Fanuc TP program (LS listing): btu_logo.ls

/PROG  btu_logo
/ATTR
COMMENT	= "19-03-22 13:07:40";
PROG_SIZE	= 0;
DEFAULT_GROUP	= 1, *, *, *, *;
/APPL
    ARC Welding Equipment: 1, *, *, *, *;
/MN
   1:  CALL HOME_ALL;
   1:  UFRAME_NUM = 1;
   1:  UTOOL_NUM = 3;
   1:  COL GUARD ADJUST 150;
   1:  MESSAGE[- Layer/Ebene 1];
   1:  PR[91] = PR[90];
   1:  GO[2]=3;
   1:  PR[91,1] = PR[90,1] + 3.907;
   1:  PR[91,2] = PR[90,2] + 46.803;
   1:  PR[91,3] = PR[90,3] + 2.795;
   1:  MESSAGE[Teach Startpoint in PR91];
   1:  MESSAGE[Weld speed R100 in mm/sec];
   1:  MESSAGE[Retraction +Z in R101 in mm];
   1:  MESSAGE[Retraction speed in R102 in %];
   1:  PR[92] = PR[91];
   1:  PR[92,3] = PR[92,3] + R[101];
   1:J PR[92] R[102]% CNT100;
   1:L PR[91] 100mm/sec CNT100 RampTo R[100];
   1:  PR[91,1] = PR[90,1] + 3.583;
   1:  PR[91,2] = PR[90,2] + 46.861;
   1:L PR[91] R[100]mm/sec CNT100;
   1:  PR[91,1] = PR[90,1] + 3.247;
   1:  PR[91,2] = PR[90,2] + 46.900;
   1:L PR[91] R[100]mm/sec CNT100;
   1:  PR[91,1] = PR[90,1] + 2.612;
   1:  PR[91,2] = PR[90,2] + 47.029;
   1:L PR[91] R[100]mm/sec CNT100;
   1:  PR[91,1] = PR[90,1] + 1.805;
   1:  PR[91,2] = PR[90,2] + 47.067;
   1:L PR[91] R[100]mm/sec CNT100;
   1:  PR[91,1] = PR[90,1] + 1.782;
   1:  PR[91,2] = PR[90,2] + 47.066;
   1:L PR[91] R[100]mm/sec CNT100;
   1:  PR[91,1] = PR[90,1] + 1.030;
   1:  PR[91,2] = PR[90,2] + 46.980;
   1:L PR[91] R[100]mm/sec CNT100;
   1:  PR[91,1] = PR[90,1] + 0.258;
   1:  PR[91,2] = PR[90,2] + 46.814;
   1:L PR[91] R[100]mm/sec CNT100;
   1:  PR[91,1] = PR[90,1] + -0.573;
   1:  PR[91,2] = PR[90,2] + 46.433;
   1:L PR[91] R[100]mm/sec CNT100;
   1:  PR[91,1] = PR[90,1] + -0.582;
   1:  PR[91,2] = PR[90,2] + 46.430;
   1:L PR[91] R[100]mm/sec CNT100;
   1:  PR[91,1] = PR[90,1] + -1.294;
   1:  PR[91,2] = PR[90,2] + 45.950;
   1:L PR[91] R[100]mm/sec CNT100;
   1:  PR[91,1] = PR[90,1] + -1.634;
   1:  PR[91,2] = PR[90,2] + 45.636;
   1:L PR[91] R[100]mm/sec CNT100;
   1:  PR[91,1] = PR[90,1] + -2.312;
   1:  PR[91,2] = PR[90,2] + 44.852;
   1:L PR[91] R[100]mm/sec CNT100;
   1:  PR[91,1] = PR[90,1] + -2.541;
   1:  PR[91,2] = PR[90,2] + 44.349;
   1:L PR[91] R[100]mm/sec CNT100;
   1:  PR[91,1] = PR[90,1] + -2.727;
   1:  PR[91,2] = PR[90,2] + 43.996;
   1:L PR[91] R[100]mm/sec CNT100;
   1:  PR[91,1] = PR[90,1] + -3.065;
   1:  PR[91,2] = PR[90,2] + 43.254;
   1:L PR[91] R[100]mm/sec CNT100;
   1:  PR[91,1] = PR[90,1] + -3.083;
   1:  PR[91,2] = PR[90,2] + 43.063;
   1:L PR[91] R[100]mm/sec CNT100;
   1:  PR[91,1] = PR[90,1] + -3.240;
   1:  PR[91,2] = PR[90,2] + 42.434;
   1:L PR[91] R[100]mm/sec CNT100;
   1:  PR[91,1] = PR[90,1] + -3.248;
   1:  PR[91,2] = PR[90,2] + 42.049;
   1:L PR[91] R[100]mm/sec CNT100;
   1:  PR[91,1] = PR[90,1] + -3.284;
   1:  PR[91,2] = PR[90,2] + 41.564;
   1:L PR[91] R[100]mm/sec CNT100;
   1:  PR[91,1] = PR[90,1] + -3.289;
   1:  PR[91,2] = PR[90,2] + 40.607;
   1:L PR[91] R[100]mm/sec CNT100;
   1:  PR[91,1] = PR[90,1] + -3.286;
   1:  PR[91,2] = PR[90,2] + 2.178;
   1:L PR[91] R[100]mm/sec CNT100;
   1:  PR[91,1] = PR[90,1] + -3.273;
   1:  PR[91,2] = PR[90,2] + 1.199;
   1:L PR[91] R[100]mm/sec CNT100;
   1:  PR[91,1] = PR[90,1] + -3.212;
   1:  PR[91,2] = PR[90,2] + -0.213;
   1:L PR[91] R[100]mm/sec CNT100;
   1:  PR[91,1] = PR[90,1] + -3.152;
   1:  PR[91,2] = PR[90,2] + -0.737;
   1:L PR[91] R[100]mm/sec CNT100;
   1:  PR[91,1] = PR[90,1] + -3.131;
   1:  PR[91,2] = PR[90,2] + -1.080;
   1:L PR[91] R[100]mm/sec CNT100;
   1:  PR[91,1] = PR[90,1] + -3.026;
   1:  PR[91,2] = PR[90,2] + -1.687;
   1:L PR[91] R[100]mm/sec CNT100;
   1:  PR[91,1] = PR[90,1] + -3.009;
   1:  PR[91,2] = PR[90,2] + -1.889;
   1:L PR[91] R[100]mm/sec CNT100;
   1:  PR[91,1] = PR[90,1] + -2.860;
   1:  PR[91,2] = PR[90,2] + -2.483;
   1:L PR[91] R[100]mm/sec CNT100;
   1:  PR[91,1] = PR[90,1] + -2.816;
   1:  PR[91,2] = PR[90,2] + -2.594;
   1:L PR[91] R[100]mm/sec CNT100;
   1:  PR[91,1] = PR[90,1] + -2.568;
   1:  PR[91,2] = PR[90,2] + -3.464;
   1:L PR[91] R[100]mm/sec CNT100;
   1:  PR[91,1] = PR[90,1] + -2.555;
   1:  PR[91,2] = PR[90,2] + -3.686;
   1:L PR[91] R[100]mm/sec CNT100;
   1:  PR[91,1] = PR[90,1] + -2.415;
   1:  PR[91,2] = PR[90,2] + -4.292;
   1:L PR[91] R[100]mm/sec CNT100;
   1:  PR[91,1] = PR[90,1] + -2.298;
   1:  PR[91,2] = PR[90,2] + -5.127;
   1:L PR[91] R[100]mm/sec CNT100;
   1:  PR[91,1] = PR[90,1] + -2.153;
   1:  PR[91,2] = PR[90,2] + -5.601;
   1:L PR[91] R[100]mm/sec CNT100;
   1:  PR[91,1] = PR[90,1] + -2.125;
   1:  PR[91,2] = PR[90,2] + -5.801;
   1:L PR[91] R[100]mm/sec CNT100;
   1:  PR[91,1] = PR[90,1] + -1.883;
   1:  PR[91,2] = PR[90,2] + -6.260;
   1:L PR[91] R[100]mm/sec CNT100;
   1:  PR[91,1] = PR[90,1] + -1.467;
   1:  PR[91,2] = PR[90,2] + -7.196;
   1:L PR[91] R[100]mm/sec CNT100;
   1:  PR[91,1] = PR[90,1] + -1.390;
   1:  PR[91,2] = PR[90,2] + -7.658;
   1:L PR[91] R[100]mm/sec CNT100;
   1:  PR[91,1] = PR[90,1] + -1.315;
   1:  PR[91,2] = PR[90,2] + -7.984;
   1:L PR[91] R[100]mm/sec CNT100;
   1:  PR[91,1] = PR[90,1] + -1.076;
   1:  PR[91,2] = PR[90,2] + -8.509;
   1:L PR[91] R[100]mm/sec CNT100;
   1:  PR[91,1] = PR[90,1] + -0.590;
   1:  PR[91,2] = PR[90,2] + -9.123;
   1:L PR[91] R[100]mm/sec CNT100;
   1:  PR[91,1] = PR[90,1] + -0.511;
   1:  PR[91,2] = PR[90,2] + -9.599;
   1:L PR[91] R[100]mm/sec CNT100;
   1:  PR[91,1] = PR[90,1] + -0.388;
   1:  PR[91,2] = PR[90,2] + -9.951;
   1:L PR[91] R[100]mm/sec CNT100;
   1:  PR[91,1] = PR[90,1] + -0.146;
   1:  PR[91,2] = PR[90,2] + -10.451;
   1:L PR[91] R[100]mm/sec CNT100;
   1:  PR[91,1] = PR[90,1] + 0.394;
   1:  PR[91,2] = PR[90,2] + -11.007;
   1:L PR[91] R[100]mm/sec CNT100;
   1:  PR[91,1] = PR[90,1] + 0.519;
   1:  PR[91,2] = PR[90,2] + -11.563;
   1:L PR[91] R[100]mm/sec CNT100;
   1:  PR[91,1] = PR[90,1] + 0.605;
   1:  PR[91,2] = PR[90,2] + -11.789;
   1:L PR[91] R[100]mm/sec CNT100;
   1:  PR[91,1] = PR[90,1] + 0.908;
   1:  PR[91,2] = PR[90,2] + -12.207;
   1:L PR[91] R[100]mm/sec CNT100;
   1:  PR[91,1] = PR[90,1] + 1.443;
   1:  PR[91,2] = PR[90,2] + -12.862;
   1:L PR[91] R[100]mm/sec CNT100;
   1:  PR[91,1] = PR[90,1] + 1.693;
   1:  PR[91,2] = PR[90,2] + -13.439;
   1:L PR[91] R[100]mm/sec CNT100;
   1:  PR[91,1] = PR[90,1] + 2.296;
   1:  PR[91,2] = PR[90,2] + -13.860;
   1:L PR[91] R[100]mm/sec CNT100;
   1:  PR[91,1] = PR[90,1] + 2.491;
   1:  PR[91,2] = PR[90,2] + -14.478;
   1:L PR[91] R[100]mm/sec CNT100;
   1:  PR[91,1] = PR[90,1] + 2.535;
   1:  PR[91,2] = PR[90,2] + -14.568;
   1:L PR[91] R[100]mm/sec CNT100;
   1:  PR[91,1] = PR[90,1] + 2.606;
   1:  PR[91,2] = PR[90,2] + -14.628;
   1:L PR[91] R[100]mm/sec CNT100;
   1:  PR[91,1] = PR[90,1] + 3.140;
   1:  PR[91,2] = PR[90,2] + -14.874;
   1:L PR[91] R[100]mm/sec CNT100;
   1:  PR[91,1] = PR[90,1] + 3.291;
   1:  PR[91,2] = PR[90,2] + -15.406;
   1:L PR[91] R[100]mm/sec CNT100;
   1:  PR[91,1] = PR[90,1] + 3.418;
   1:  PR[91,2] = PR[90,2] + -15.595;
   1:L PR[91] R[100]mm/sec CNT100;
   1:  PR[91,1] = PR[90,1] + 3.876;
   1:  PR[91,2] = PR[90,2] + -16.020;
   1:L PR[91] R[100]mm/sec CNT100;
   1:  PR[91,1] = PR[90,1] + 4.332;
   1:  PR[91,2] = PR[90,2] + -16.568;
   1:L PR[91] R[100]mm/sec CNT100;
   1:  PR[91,1] = PR[90,1] + 4.569;
   1:  PR[91,2] = PR[90,2] + -16.781;
   1:L PR[91] R[100]mm/sec CNT100;
   1:  PR[91,1] = PR[90,1] + 4.637;
   1:  PR[91,2] = PR[90,2] + -16.802;
   1:L PR[91] R[100]mm/sec CNT100;
   1:  PR[91,1] = PR[90,1] + 4.837;
   1:  PR[91,2] = PR[90,2] + -17.021;
   1:L PR[91] R[100]mm/sec CNT100;
   1:  PR[91,1] = PR[90,1] + 5.058;
   1:  PR[91,2] = PR[90,2] + -17.219;
   1:L PR[91] R[100]mm/sec CNT100;
   1:  PR[91,1] = PR[90,1] + 5.080;
   1:  PR[91,2] = PR[90,2] + -17.287;
   1:L PR[91] R[100]mm/sec CNT100;
   1:  PR[91,1] = PR[90,1] + 5.278;
   1:  PR[91,2] = PR[90,2] + -17.504;
   1:L PR[91] R[100]mm/sec CNT100;
   1:  PR[91,1] = PR[90,1] + 5.496;
   1:  PR[91,2] = PR[90,2] + -17.670;
   1:L PR[91] R[100]mm/sec CNT100;
   1:  PR[91,1] = PR[90,1] + 5.968;
   1:  PR[91,2] = PR[90,2] + -17.809;
   1:L PR[91] R[100]mm/sec CNT100;
   1:  PR[91,1] = PR[90,1] + 6.157;
   1:  PR[91,2] = PR[90,2] + -18.284;
   1:L PR[91] R[100]mm/sec CNT100;
   1:  PR[91,1] = PR[90,1] + 6.273;
   1:  PR[91,2] = PR[90,2] + -18.417;
   1:L PR[91] R[100]mm/sec CNT100;
   1:  PR[91,1] = PR[90,1] + 6.417;
   1:  PR[91,2] = PR[90,2] + -18.501;
   1:L PR[91] R[100]mm/sec CNT100;
   1:  PR[91,1] = PR[90,1] + 6.992;
   1:  PR[91,2] = PR[90,2] + -18.676;
   1:L PR[91] R[100]mm/sec CNT100;
   1:  PR[91,1] = PR[90,1] + 7.313;
   1:  PR[91,2] = PR[90,2] + -19.266;
   1:L PR[91] R[100]mm/sec CNT100;
   1:  PR[91,1] = PR[90,1] + 7.323;
   1:  PR[91,2] = PR[90,2] + -19.279;
   1:L PR[91] R[100]mm/sec CNT100;
   1:  PR[91,1] = PR[90,1] + 7.984;
   1:  PR[91,2] = PR[90,2] + -19.542;
   1:L PR[91] R[100]mm/sec CNT100;
   1:  PR[91,1] = PR[90,1] + 8.501;
   1:  PR[91,2] = PR[90,2] + -20.109;
   1:L PR[91] R[100]mm/sec CNT100;
   1:  PR[91,1] = PR[90,1] + 9.363;
   1:  PR[91,2] = PR[90,2] + -20.602;
   1:L PR[91] R[100]mm/sec CNT100;
   1:  PR[91,1] = PR[90,1] + 9.775;
   1:  PR[91,2] = PR[90,2] + -20.686;
   1:L PR[91] R[100]mm/sec CNT100;
   1:  PR[91,1] = PR[90,1] + 10.086;
   1:  PR[91,2] = PR[90,2] + -21.118;
   1:L PR[91] R[100]mm/sec CNT100;
   1:  PR[91,1] = PR[90,1] + 10.181;
   1:  PR[91,2] = PR[90,2] + -21.207;
   1:L PR[91] R[100]mm/sec CNT100;
   1:  PR[91,1] = PR[90,1] + 10.801;
   1:  PR[91,2] = PR[90,2] + -21.397;
   1:L PR[91] R[100]mm/sec CNT100;
   1:  PR[91,1] = PR[90,1] + 11.399;
   1:  PR[91,2] = PR[90,2] + -21.763;
   1:L PR[91] R[100]mm/sec CNT100;
   1:  PR[91,1] = PR[90,1] + 11.435;
   1:  PR[91,2] = PR[90,2] + -21.770;
   1:L PR[91] R[100]mm/sec CNT100;
   1:  PR[91,1] = PR[90,1] + 11.604;
   1:  PR[91,2] = PR[90,2] + -21.889;
   1:L PR[91] R[100]mm/sec CNT100;
   1:  PR[91,1] = PR[90,1] + 11.768;
   1:  PR[91,2] = PR[90,2] + -21.989;
   1:L PR[91] R[100]mm/sec CNT100;
   1:  PR[91,1] = PR[90,1] + 11.793;
   1:  PR[91,2] = PR[90,2] + -22.021;
   1:L PR[91] R[100]mm/sec CNT100;
   1:  PR[91,1] = PR[90,1] + 12.031;
   1:  PR[91,2] = PR[90,2] + -22.189;
   1:L PR[91] R[100]mm/sec CNT100;
   1:  PR[91,1] = PR[90,1] + 12.693;
   1:  PR[91,2] = PR[90,2] + -22.356;
   1:L PR[91] R[100]mm/sec CNT100;
   1:  PR[91,1] = PR[90,1] + 13.271;
   1:  PR[91,2] = PR[90,2] + -22.616;
   1:L PR[91] R[100]mm/sec CNT100;
   1:  PR[91,1] = PR[90,1] + 13.463;
   1:  PR[91,2] = PR[90,2] + -22.644;
   1:L PR[91] R[100]mm/sec CNT100;
   1:  PR[91,1] = PR[90,1] + 14.077;
   1:  PR[91,2] = PR[90,2] + -23.062;
   1:L PR[91] R[100]mm/sec CNT100;
   1:  PR[91,1] = PR[90,1] + 14.229;
   1:  PR[91,2] = PR[90,2] + -23.088;
   1:L PR[91] R[100]mm/sec CNT100;
   1:  PR[91,1] = PR[90,1] + 14.701;
   1:  PR[91,2] = PR[90,2] + -23.254;
   1:L PR[91] R[100]mm/sec CNT100;
   1:  PR[91,1] = PR[90,1] + 15.107;
   1:  PR[91,2] = PR[90,2] + -23.339;
   1:L PR[91] R[100]mm/sec CNT100;
   1:  PR[91,1] = PR[90,1] + 15.505;
   1:  PR[91,2] = PR[90,2] + -23.390;
   1:L PR[91] R[100]mm/sec CNT100;
   1:  PR[91,1] = PR[90,1] + 16.450;
   1:  PR[91,2] = PR[90,2] + -23.736;
   1:L PR[91] R[100]mm/sec CNT100;
   1:  PR[91,1] = PR[90,1] + 16.984;
   1:  PR[91,2] = PR[90,2] + -23.975;
   1:L PR[91] R[100]mm/sec CNT100;
   1:  PR[91,1] = PR[90,1] + 17.171;
   1:  PR[91,2] = PR[90,2] + -23.997;
   1:L PR[91] R[100]mm/sec CNT100;
   1:  PR[91,1] = PR[90,1] + 17.682;
   1:  PR[91,2] = PR[90,2] + -24.148;
   1:L PR[91] R[100]mm/sec CNT100;
   1:  PR[91,1] = PR[90,1] + 18.072;
   1:  PR[91,2] = PR[90,2] + -24.185;
   1:L PR[91] R[100]mm/sec CNT100;
   1:  PR[91,1] = PR[90,1] + 18.481;
   1:  PR[91,2] = PR[90,2] + -24.256;
   1:L PR[91] R[100]mm/sec CNT100;
   1:  PR[91,1] = PR[90,1] + 19.386;
   1:  PR[91,2] = PR[90,2] + -24.338;
   1:L PR[91] R[100]mm/sec CNT100;
   1:  PR[91,1] = PR[90,1] + 20.021;
   1:  PR[91,2] = PR[90,2] + -24.433;
   1:L PR[91] R[100]mm/sec CNT100;
   1:  PR[91,1] = PR[90,1] + 20.235;
   1:  PR[91,2] = PR[90,2] + -24.441;
   1:L PR[91] R[100]mm/sec CNT100;
   1:  PR[91,1] = PR[90,1] + 21.062;
   1:  PR[91,2] = PR[90,2] + -24.556;
   1:L PR[91] R[100]mm/sec CNT100;
   1:  PR[91,1] = PR[90,1] + 22.010;
   1:  PR[91,2] = PR[90,2] + -24.647;
   1:L PR[91] R[100]mm/sec CNT100;
   1:  PR[91,1] = PR[90,1] + 22.916;
   1:  PR[91,2] = PR[90,2] + -24.702;
   1:L PR[91] R[100]mm/sec CNT100;
   1:  PR[91,1] = PR[90,1] + 23.747;
   1:  PR[91,2] = PR[90,2] + -24.671;
   1:L PR[91] R[100]mm/sec CNT100;
   1:  PR[91,1] = PR[90,1] + 24.799;
   1:  PR[91,2] = PR[90,2] + -24.489;
   1:L PR[91] R[100]mm/sec CNT100;
   1:  PR[91,1] = PR[90,1] + 25.392;
   1:  PR[91,2] = PR[90,2] + -24.342;
   1:L PR[91] R[100]mm/sec CNT100;
   1:  PR[91,1] = PR[90,1] + 26.153;
   1:  PR[91,2] = PR[90,2] + -23.964;
   1:L PR[91] R[100]mm/sec CNT100;
   1:  PR[91,1] = PR[90,1] + 26.227;
   1:  PR[91,2] = PR[90,2] + -23.942;
   1:L PR[91] R[100]mm/sec CNT100;
   1:  PR[91,1] = PR[90,1] + 26.236;
   1:  PR[91,2] = PR[90,2] + -23.935;
   1:L PR[91] R[100]mm/sec CNT100;
   1:  PR[91,1] = PR[90,1] + 26.967;
   1:  PR[91,2] = PR[90,2] + -23.430;
   1:L PR[91] R[100]mm/sec CNT100;
   1:  PR[91,1] = PR[90,1] + 27.290;
   1:  PR[91,2] = PR[90,2] + -23.116;
   1:L PR[91] R[100]mm/sec CNT100;
   1:  PR[91,1] = PR[90,1] + 27.934;
   1:  PR[91,2] = PR[90,2] + -22.343;
   1:L PR[91] R[100]mm/sec CNT100;
   1:  PR[91,1] = PR[90,1] + 28.078;
   1:  PR[91,2] = PR[90,2] + -21.991;
   1:L PR[91] R[100]mm/sec CNT100;
   1:  PR[91,1] = PR[90,1] + 28.310;
   1:  PR[91,2] = PR[90,2] + -21.508;
   1:L PR[91] R[100]mm/sec CNT100;
   1:  PR[91,1] = PR[90,1] + 28.560;
   1:  PR[91,2] = PR[90,2] + -20.886;
   1:L PR[91] R[100]mm/sec CNT100;
   1:  PR[91,1] = PR[90,1] + 28.642;
   1:  PR[91,2] = PR[90,2] + -20.714;
   1:L PR[91] R[100]mm/sec CNT100;
   1:  PR[91,1] = PR[90,1] + 28.644;
   1:  PR[91,2] = PR[90,2] + -20.690;
   1:L PR[91] R[100]mm/sec CNT100;
   1:  PR[91,1] = PR[90,1] + 28.814;
   1:  PR[91,2] = PR[90,2] + -19.912;
   1:L PR[91] R[100]mm/sec CNT100;
   1:  PR[91,1] = PR[90,1] + 28.832;
   1:  PR[91,2] = PR[90,2] + -19.085;
   1:L PR[91] R[100]mm/sec CNT100;
   1:  PR[91,1] = PR[90,1] + 28.825;
   1:  PR[91,2] = PR[90,2] + -18.855;
   1:L PR[91] R[100]mm/sec CNT100;
   1:  PR[91,1] = PR[90,1] + 28.717;
   1:  PR[91,2] = PR[90,2] + -18.298;
   1:L PR[91] R[100]mm/sec CNT100;
   1:  PR[91,1] = PR[90,1] + 28.602;
   1:  PR[91,2] = PR[90,2] + -18.109;
   1:L PR[91] R[100]mm/sec CNT100;
   1:  PR[91,1] = PR[90,1] + 28.370;
   1:  PR[91,2] = PR[90,2] + -17.589;
   1:L PR[91] R[100]mm/sec CNT100;
   1:  PR[91,1] = PR[90,1] + 28.350;
   1:  PR[91,2] = PR[90,2] + -17.451;
   1:L PR[91] R[100]mm/sec CNT100;
   1:  PR[91,1] = PR[90,1] + 28.003;
   1:  PR[91,2] = PR[90,2] + -16.589;
   1:L PR[91] R[100]mm/sec CNT100;
   1:  PR[91,1] = PR[90,1] + 27.500;
   1:  PR[91,2] = PR[90,2] + -16.147;
   1:L PR[91] R[100]mm/sec CNT100;
   1:  PR[91,1] = PR[90,1] + 27.277;
   1:  PR[91,2] = PR[90,2] + -15.662;
   1:L PR[91] R[100]mm/sec CNT100;
   1:  PR[91,1] = PR[90,1] + 26.782;
   1:  PR[91,2] = PR[90,2] + -15.428;
   1:L PR[91] R[100]mm/sec CNT100;
   1:  PR[91,1] = PR[90,1] + 26.375;
   1:  PR[91,2] = PR[90,2] + -14.932;
   1:L PR[91] R[100]mm/sec CNT100;
   1:  PR[91,1] = PR[90,1] + 25.497;
   1:  PR[91,2] = PR[90,2] + -14.558;
   1:L PR[91] R[100]mm/sec CNT100;
   1:  PR[91,1] = PR[90,1] + 25.382;
   1:  PR[91,2] = PR[90,2] + -14.540;
   1:L PR[91] R[100]mm/sec CNT100;
   1:  PR[91,1] = PR[90,1] + 24.952;
   1:  PR[91,2] = PR[90,2] + -14.335;
   1:L PR[91] R[100]mm/sec CNT100;
   1:  PR[91,1] = PR[90,1] + 24.711;
   1:  PR[91,2] = PR[90,2] + -14.194;
   1:L PR[91] R[100]mm/sec CNT100;
   1:  PR[91,1] = PR[90,1] + 24.683;
   1:  PR[91,2] = PR[90,2] + -14.191;
   1:L PR[91] R[100]mm/sec CNT100;
   1:  PR[91,1] = PR[90,1] + 24.124;
   1:  PR[91,2] = PR[90,2] + -14.075;
   1:L PR[91] R[100]mm/sec CNT100;
   1:  PR[91,1] = PR[90,1] + 23.311;
   1:  PR[91,2] = PR[90,2] + -14.026;
   1:L PR[91] R[100]mm/sec CNT100;
   1:  PR[91,1] = PR[90,1] + 22.811;
   1:  PR[91,2] = PR[90,2] + -14.013;
   1:L PR[91] R[100]mm/sec CNT100;
   1:  PR[91,1] = PR[90,1] + 22.335;
   1:  PR[91,2] = PR[90,2] + -13.970;
   1:L PR[91] R[100]mm/sec CNT100;
   1:  PR[91,1] = PR[90,1] + 21.794;
   1:  PR[91,2] = PR[90,2] + -13.954;
   1:L PR[91] R[100]mm/sec CNT100;
   1:  PR[91,1] = PR[90,1] + 20.316;
   1:  PR[91,2] = PR[90,2] + -13.802;
   1:L PR[91] R[100]mm/sec CNT100;
   1:  PR[91,1] = PR[90,1] + 19.619;
   1:  PR[91,2] = PR[90,2] + -13.638;
   1:L PR[91] R[100]mm/sec CNT100;
   1:  PR[91,1] = PR[90,1] + 19.336;
   1:  PR[91,2] = PR[90,2] + -13.603;
   1:L PR[91] R[100]mm/sec CNT100;
   1:  PR[91,1] = PR[90,1] + 18.693;
   1:  PR[91,2] = PR[90,2] + -13.319;
   1:L PR[91] R[100]mm/sec CNT100;
   1:  PR[91,1] = PR[90,1] + 18.559;
   1:  PR[91,2] = PR[90,2] + -13.231;
   1:L PR[91] R[100]mm/sec CNT100;
   1:  PR[91,1] = PR[90,1] + 18.424;
   1:  PR[91,2] = PR[90,2] + -13.214;
   1:L PR[91] R[100]mm/sec CNT100;
   1:  PR[91,1] = PR[90,1] + 17.895;
   1:  PR[91,2] = PR[90,2] + -12.938;
   1:L PR[91] R[100]mm/sec CNT100;
   1:  PR[91,1] = PR[90,1] + 17.545;
   1:  PR[91,2] = PR[90,2] + -12.883;
   1:L PR[91] R[100]mm/sec CNT100;
   1:  PR[91,1] = PR[90,1] + 17.006;
   1:  PR[91,2] = PR[90,2] + -12.726;
   1:L PR[91] R[100]mm/sec CNT100;
   1:  PR[91,1] = PR[90,1] + 16.000;
   1:  PR[91,2] = PR[90,2] + -12.250;
   1:L PR[91] R[100]mm/sec CNT100;
   1:  PR[91,1] = PR[90,1] + 15.594;
   1:  PR[91,2] = PR[90,2] + -11.867;
   1:L PR[91] R[100]mm/sec CNT100;
   1:  PR[91,1] = PR[90,1] + 15.397;
   1:  PR[91,2] = PR[90,2] + -11.818;
   1:L PR[91] R[100]mm/sec CNT100;
   1:  PR[91,1] = PR[90,1] + 14.787;
   1:  PR[91,2] = PR[90,2] + -11.570;
   1:L PR[91] R[100]mm/sec CNT100;
   1:  PR[91,1] = PR[90,1] + 14.179;
   1:  PR[91,2] = PR[90,2] + -11.063;
   1:L PR[91] R[100]mm/sec CNT100;
   1:  PR[91,1] = PR[90,1] + 13.571;
   1:  PR[91,2] = PR[90,2] + -10.569;
   1:L PR[91] R[100]mm/sec CNT100;
   1:  PR[91,1] = PR[90,1] + 12.825;
   1:  PR[91,2] = PR[90,2] + -10.073;
   1:L PR[91] R[100]mm/sec CNT100;
   1:  PR[91,1] = PR[90,1] + 12.382;
   1:  PR[91,2] = PR[90,2] + -9.498;
   1:L PR[91] R[100]mm/sec CNT100;
   1:  PR[91,1] = PR[90,1] + 11.707;
   1:  PR[91,2] = PR[90,2] + -9.050;
   1:L PR[91] R[100]mm/sec CNT100;
   1:  PR[91,1] = PR[90,1] + 11.257;
   1:  PR[91,2] = PR[90,2] + -8.315;
   1:L PR[91] R[100]mm/sec CNT100;
   1:  PR[91,1] = PR[90,1] + 10.951;
   1:  PR[91,2] = PR[90,2] + -8.029;
   1:L PR[91] R[100]mm/sec CNT100;
   1:  PR[91,1] = PR[90,1] + 10.858;
   1:  PR[91,2] = PR[90,2] + -7.989;
   1:L PR[91] R[100]mm/sec CNT100;
   1:  PR[91,1] = PR[90,1] + 10.763;
   1:  PR[91,2] = PR[90,2] + -7.854;
   1:L PR[91] R[100]mm/sec CNT100;
   1:  PR[91,1] = PR[90,1] + 10.639;
   1:  PR[91,2] = PR[90,2] + -7.738;
   1:L PR[91] R[100]mm/sec CNT100;
   1:  PR[91,1] = PR[90,1] + 10.613;
   1:  PR[91,2] = PR[90,2] + -7.641;
   1:L PR[91] R[100]mm/sec CNT100;
   1:  PR[91,1] = PR[90,1] + 10.227;
   1:  PR[91,2] = PR[90,2] + -7.091;
   1:L PR[91] R[100]mm/sec CNT100;
   1:  PR[91,1] = PR[90,1] + 9.869;
   1:  PR[91,2] = PR[90,2] + -6.478;
   1:L PR[91] R[100]mm/sec CNT100;
   1:  PR[91,1] = PR[90,1] + 9.865;
   1:  PR[91,2] = PR[90,2] + -6.460;
   1:L PR[91] R[100]mm/sec CNT100;
   1:  PR[91,1] = PR[90,1] + 9.309;
   1:  PR[91,2] = PR[90,2] + -5.884;
   1:L PR[91] R[100]mm/sec CNT100;
   1:  PR[91,1] = PR[90,1] + 9.024;
   1:  PR[91,2] = PR[90,2] + -4.910;
   1:L PR[91] R[100]mm/sec CNT100;
   1:  PR[91,1] = PR[90,1] + 8.736;
   1:  PR[91,2] = PR[90,2] + -4.394;
   1:L PR[91] R[100]mm/sec CNT100;
   1:  PR[91,1] = PR[90,1] + 8.720;
   1:  PR[91,2] = PR[90,2] + -4.284;
   1:L PR[91] R[100]mm/sec CNT100;
   1:  PR[91,1] = PR[90,1] + 8.645;
   1:  PR[91,2] = PR[90,2] + -4.205;
   1:L PR[91] R[100]mm/sec CNT100;
   1:  PR[91,1] = PR[90,1] + 8.255;
   1:  PR[91,2] = PR[90,2] + -3.596;
   1:L PR[91] R[100]mm/sec CNT100;
   1:  PR[91,1] = PR[90,1] + 8.191;
   1:  PR[91,2] = PR[90,2] + -3.224;
   1:L PR[91] R[100]mm/sec CNT100;
   1:  PR[91,1] = PR[90,1] + 8.017;
   1:  PR[91,2] = PR[90,2] + -2.611;
   1:L PR[91] R[100]mm/sec CNT100;
   1:  PR[91,1] = PR[90,1] + 7.906;
   1:  PR[91,2] = PR[90,2] + -2.112;
   1:L PR[91] R[100]mm/sec CNT100;
   1:  PR[91,1] = PR[90,1] + 7.864;
   1:  PR[91,2] = PR[90,2] + -1.663;
   1:L PR[91] R[100]mm/sec CNT100;
   1:  PR[91,1] = PR[90,1] + 7.698;
   1:  PR[91,2] = PR[90,2] + -1.148;
   1:L PR[91] R[100]mm/sec CNT100;
   1:  PR[91,1] = PR[90,1] + 7.676;
   1:  PR[91,2] = PR[90,2] + -0.789;
   1:L PR[91] R[100]mm/sec CNT100;
   1:  PR[91,1] = PR[90,1] + 7.477;
   1:  PR[91,2] = PR[90,2] + -0.103;
   1:L PR[91] R[100]mm/sec CNT100;
   1:  PR[91,1] = PR[90,1] + 7.467;
   1:  PR[91,2] = PR[90,2] + 0.101;
   1:L PR[91] R[100]mm/sec CNT100;
   1:  PR[91,1] = PR[90,1] + 7.307;
   1:  PR[91,2] = PR[90,2] + 0.934;
   1:L PR[91] R[100]mm/sec CNT100;
   1:  PR[91,1] = PR[90,1] + 7.236;
   1:  PR[91,2] = PR[90,2] + 2.012;
   1:L PR[91] R[100]mm/sec CNT100;
   1:  PR[91,1] = PR[90,1] + 7.217;
   1:  PR[91,2] = PR[90,2] + 3.055;
   1:L PR[91] R[100]mm/sec CNT100;
   1:  PR[91,1] = PR[90,1] + 7.214;
   1:  PR[91,2] = PR[90,2] + 15.414;
   1:L PR[91] R[100]mm/sec CNT100;
   1:  PR[91,1] = PR[90,1] + 7.350;
   1:  PR[91,2] = PR[90,2] + 16.486;
   1:L PR[91] R[100]mm/sec CNT100;
   1:  PR[91,1] = PR[90,1] + 7.530;
   1:  PR[91,2] = PR[90,2] + 17.240;
   1:L PR[91] R[100]mm/sec CNT100;
   1:  PR[91,1] = PR[90,1] + 9.293;
   1:  PR[91,2] = PR[90,2] + 18.453;
   1:L PR[91] R[100]mm/sec CNT100;
   1:  PR[91,1] = PR[90,1] + 10.734;
   1:  PR[91,2] = PR[90,2] + 18.613;
   1:L PR[91] R[100]mm/sec CNT100;
   1:  PR[91,1] = PR[90,1] + 11.821;
   1:  PR[91,2] = PR[90,2] + 18.642;
   1:L PR[91] R[100]mm/sec CNT100;
   1:  PR[91,1] = PR[90,1] + 22.856;
   1:  PR[91,2] = PR[90,2] + 18.657;
   1:L PR[91] R[100]mm/sec CNT100;
   1:  PR[91,1] = PR[90,1] + 23.697;
   1:  PR[91,2] = PR[90,2] + 18.703;
   1:L PR[91] R[100]mm/sec CNT100;
   1:  PR[91,1] = PR[90,1] + 24.187;
   1:  PR[91,2] = PR[90,2] + 18.812;
   1:L PR[91] R[100]mm/sec CNT100;
   1:  PR[91,1] = PR[90,1] + 24.667;
   1:  PR[91,2] = PR[90,2] + 18.901;
   1:L PR[91] R[100]mm/sec CNT100;
   1:  PR[91,1] = PR[90,1] + 25.385;
   1:  PR[91,2] = PR[90,2] + 19.098;
   1:L PR[91] R[100]mm/sec CNT100;
   1:  PR[91,1] = PR[90,1] + 26.017;
   1:  PR[91,2] = PR[90,2] + 19.403;
   1:L PR[91] R[100]mm/sec CNT100;
   1:  PR[91,1] = PR[90,1] + 26.230;
   1:  PR[91,2] = PR[90,2] + 19.470;
   1:L PR[91] R[100]mm/sec CNT100;
   1:  PR[91,1] = PR[90,1] + 26.951;
   1:  PR[91,2] = PR[90,2] + 20.000;
   1:L PR[91] R[100]mm/sec CNT100;
   1:  PR[91,1] = PR[90,1] + 27.351;
   1:  PR[91,2] = PR[90,2] + 20.390;
   1:L PR[91] R[100]mm/sec CNT100;
   1:  PR[91,1] = PR[90,1] + 27.765;
   1:  PR[91,2] = PR[90,2] + 20.880;
   1:L PR[91] R[100]mm/sec CNT100;
   1:  PR[91,1] = PR[90,1] + 27.979;
   1:  PR[91,2] = PR[90,2] + 21.152;
   1:L PR[91] R[100]mm/sec CNT100;
   1:  PR[91,1] = PR[90,1] + 28.331;
   1:  PR[91,2] = PR[90,2] + 21.966;
   1:L PR[91] R[100]mm/sec CNT100;
   1:  PR[91,1] = PR[90,1] + 28.554;
   1:  PR[91,2] = PR[90,2] + 22.523;
   1:L PR[91] R[100]mm/sec CNT100;
   1:  PR[91,1] = PR[90,1] + 28.668;
   1:  PR[91,2] = PR[90,2] + 22.770;
   1:L PR[91] R[100]mm/sec CNT100;
   1:  PR[91,1] = PR[90,1] + 28.671;
   1:  PR[91,2] = PR[90,2] + 22.825;
   1:L PR[91] R[100]mm/sec CNT100;
   1:  PR[91,1] = PR[90,1] + 28.821;
   1:  PR[91,2] = PR[90,2] + 23.569;
   1:L PR[91] R[100]mm/sec CNT100;
   1:  PR[91,1] = PR[90,1] + 28.828;
   1:  PR[91,2] = PR[90,2] + 24.405;
   1:L PR[91] R[100]mm/sec CNT100;
   1:  PR[91,1] = PR[90,1] + 28.821;
   1:  PR[91,2] = PR[90,2] + 24.623;
   1:L PR[91] R[100]mm/sec CNT100;
   1:  PR[91,1] = PR[90,1] + 28.708;
   1:  PR[91,2] = PR[90,2] + 25.141;
   1:L PR[91] R[100]mm/sec CNT100;
   1:  PR[91,1] = PR[90,1] + 28.615;
   1:  PR[91,2] = PR[90,2] + 25.282;
   1:L PR[91] R[100]mm/sec CNT100;
   1:  PR[91,1] = PR[90,1] + 28.348;
   1:  PR[91,2] = PR[90,2] + 25.875;
   1:L PR[91] R[100]mm/sec CNT100;
   1:  PR[91,1] = PR[90,1] + 28.317;
   1:  PR[91,2] = PR[90,2] + 26.065;
   1:L PR[91] R[100]mm/sec CNT100;
   1:  PR[91,1] = PR[90,1] + 28.161;
   1:  PR[91,2] = PR[90,2] + 26.488;
   1:L PR[91] R[100]mm/sec CNT100;
   1:  PR[91,1] = PR[90,1] + 27.987;
   1:  PR[91,2] = PR[90,2] + 26.855;
   1:L PR[91] R[100]mm/sec CNT100;
   1:  PR[91,1] = PR[90,1] + 27.494;
   1:  PR[91,2] = PR[90,2] + 27.311;
   1:L PR[91] R[100]mm/sec CNT100;
   1:  PR[91,1] = PR[90,1] + 27.236;
   1:  PR[91,2] = PR[90,2] + 27.795;
   1:L PR[91] R[100]mm/sec CNT100;
   1:  PR[91,1] = PR[90,1] + 26.757;
   1:  PR[91,2] = PR[90,2] + 28.045;
   1:L PR[91] R[100]mm/sec CNT100;
   1:  PR[91,1] = PR[90,1] + 26.312;
   1:  PR[91,2] = PR[90,2] + 28.539;
   1:L PR[91] R[100]mm/sec CNT100;
   1:  PR[91,1] = PR[90,1] + 25.944;
   1:  PR[91,2] = PR[90,2] + 28.706;
   1:L PR[91] R[100]mm/sec CNT100;
   1:  PR[91,1] = PR[90,1] + 25.528;
   1:  PR[91,2] = PR[90,2] + 28.863;
   1:L PR[91] R[100]mm/sec CNT100;
   1:  PR[91,1] = PR[90,1] + 25.343;
   1:  PR[91,2] = PR[90,2] + 28.892;
   1:L PR[91] R[100]mm/sec CNT100;
   1:  PR[91,1] = PR[90,1] + 24.714;
   1:  PR[91,2] = PR[90,2] + 29.164;
   1:L PR[91] R[100]mm/sec CNT100;
   1:  PR[91,1] = PR[90,1] + 24.585;
   1:  PR[91,2] = PR[90,2] + 29.245;
   1:L PR[91] R[100]mm/sec CNT100;
   1:  PR[91,1] = PR[90,1] + 24.063;
   1:  PR[91,2] = PR[90,2] + 29.357;
   1:L PR[91] R[100]mm/sec CNT100;
   1:  PR[91,1] = PR[90,1] + 23.260;
   1:  PR[91,2] = PR[90,2] + 29.394;
   1:L PR[91] R[100]mm/sec CNT100;
   1:  PR[91,1] = PR[90,1] + 13.246;
   1:  PR[91,2] = PR[90,2] + 29.403;
   1:L PR[91] R[100]mm/sec CNT100;
   1:  PR[91,1] = PR[90,1] + 10.788;
   1:  PR[91,2] = PR[90,2] + 29.427;
   1:L PR[91] R[100]mm/sec CNT100;
   1:  PR[91,1] = PR[90,1] + 10.165;
   1:  PR[91,2] = PR[90,2] + 29.462;
   1:L PR[91] R[100]mm/sec CNT100;
   1:  PR[91,1] = PR[90,1] + 9.555;
   1:  PR[91,2] = PR[90,2] + 29.532;
   1:L PR[91] R[100]mm/sec CNT100;
   1:  PR[91,1] = PR[90,1] + 8.750;
   1:  PR[91,2] = PR[90,2] + 29.744;
   1:L PR[91] R[100]mm/sec CNT100;
   1:  PR[91,1] = PR[90,1] + 7.714;
   1:  PR[91,2] = PR[90,2] + 30.580;
   1:L PR[91] R[100]mm/sec CNT100;
   1:  PR[91,1] = PR[90,1] + 7.490;
   1:  PR[91,2] = PR[90,2] + 31.124;
   1:L PR[91] R[100]mm/sec CNT100;
   1:  PR[91,1] = PR[90,1] + 7.358;
   1:  PR[91,2] = PR[90,2] + 31.642;
   1:L PR[91] R[100]mm/sec CNT100;
   1:  PR[91,1] = PR[90,1] + 7.250;
   1:  PR[91,2] = PR[90,2] + 32.291;
   1:L PR[91] R[100]mm/sec CNT100;
   1:  PR[91,1] = PR[90,1] + 7.219;
   1:  PR[91,2] = PR[90,2] + 33.397;
   1:L PR[91] R[100]mm/sec CNT100;
   1:  PR[91,1] = PR[90,1] + 7.203;
   1:  PR[91,2] = PR[90,2] + 41.566;
   1:L PR[91] R[100]mm/sec CNT100;
   1:  PR[91,1] = PR[90,1] + 7.139;
   1:  PR[91,2] = PR[90,2] + 42.435;
   1:L PR[91] R[100]mm/sec CNT100;
   1:  PR[91,1] = PR[90,1] + 7.017;
   1:  PR[91,2] = PR[90,2] + 43.060;
   1:L PR[91] R[100]mm/sec CNT100;
   1:  PR[91,1] = PR[90,1] + 6.915;
   1:  PR[91,2] = PR[90,2] + 43.756;
   1:L PR[91] R[100]mm/sec CNT100;
   1:  PR[91,1] = PR[90,1] + 6.779;
   1:  PR[91,2] = PR[90,2] + 44.044;
   1:L PR[91] R[100]mm/sec CNT100;
   1:  PR[91,1] = PR[90,1] + 6.268;
   1:  PR[91,2] = PR[90,2] + 44.698;
   1:L PR[91] R[100]mm/sec CNT100;
   1:  PR[91,1] = PR[90,1] + 6.091;
   1:  PR[91,2] = PR[90,2] + 45.174;
   1:L PR[91] R[100]mm/sec CNT100;
   1:  PR[91,1] = PR[90,1] + 5.606;
   1:  PR[91,2] = PR[90,2] + 45.478;
   1:L PR[91] R[100]mm/sec CNT100;
   1:  PR[91,1] = PR[90,1] + 5.304;
   1:  PR[91,2] = PR[90,2] + 45.969;
   1:L PR[91] R[100]mm/sec CNT100;
   1:  PR[91,1] = PR[90,1] + 4.806;
   1:  PR[91,2] = PR[90,2] + 46.159;
   1:L PR[91] R[100]mm/sec CNT100;
   1:  PR[91,1] = PR[90,1] + 4.226;
   1:  PR[91,2] = PR[90,2] + 46.660;
   1:L PR[91] R[100]mm/sec CNT100;
   1:  PR[91,1] = PR[90,1] + 3.907;
   1:  PR[91,2] = PR[90,2] + 46.803;
   1:L PR[91] R[100]mm/sec CNT100;
   1:  PR[92] = PR[91];
   1:  PR[92,3] = PR[92,3] + R[101];
   1:J PR[92] R[102]% CNT100;
   1:  PR[91,1] = PR[90,1] + 2.300;
   1:  PR[91,2] = PR[90,2] + 44.490;
   1:  PR[92] = PR[91];
   1:  PR[92,3] = PR[92,3] + R[101];
   1:J PR[92] R[102]% CNT100;
   1:L PR[91] 100mm/sec CNT100 RampTo R[100];
   1:  PR[91,1] = PR[90,1] + -0.735;
   1:  PR[91,2] = PR[90,2] + 41.456;
   1:L PR[91] R[100]mm/sec CNT100;
   1:  PR[91,1] = PR[90,1] + -0.739;
   1:  PR[91,2] = PR[90,2] + 40.601;
   1:L PR[91] R[100]mm/sec CNT100;
   1:  PR[91,2] = PR[90,2] + 37.209;
   1:L PR[91] R[100]mm/sec CNT100;
   1:  PR[91,1] = PR[90,1] + 4.532;
   1:  PR[91,2] = PR[90,2] + 42.480;
   1:L PR[91] R[100]mm/sec CNT100;
   1:  PR[91,1] = PR[90,1] + 4.607;
   1:  PR[91,2] = PR[90,2] + 42.095;
   1:L PR[91] R[100]mm/sec CNT100;
   1:  PR[91,1] = PR[90,1] + 4.653;
   1:  PR[91,2] = PR[90,2] + 41.471;
   1:L PR[91] R[100]mm/sec CNT100;
   1:  PR[91,1] = PR[90,1] + 4.659;
   1:  PR[91,2] = PR[90,2] + 38.364;
   1:L PR[91] R[100]mm/sec CNT100;
   1:  PR[91,1] = PR[90,1] + -0.739;
   1:  PR[91,2] = PR[90,2] + 32.966;
   1:L PR[91] R[100]mm/sec CNT100;
   1:  PR[91,1] = PR[90,1] + -0.738;
   1:  PR[91,2] = PR[90,2] + 28.724;
   1:L PR[91] R[100]mm/sec CNT100;
   1:  PR[91,1] = PR[90,1] + 4.667;
   1:  PR[91,2] = PR[90,2] + 34.130;
   1:L PR[91] R[100]mm/sec CNT100;
   1:  PR[91,1] = PR[90,1] + 4.669;
   1:  PR[91,2] = PR[90,2] + 33.358;
   1:L PR[91] R[100]mm/sec CNT100;
   1:  PR[91,1] = PR[90,1] + 4.706;
   1:  PR[91,2] = PR[90,2] + 32.044;
   1:L PR[91] R[100]mm/sec CNT100;
   1:  PR[91,1] = PR[90,1] + 4.860;
   1:  PR[91,2] = PR[90,2] + 31.117;
   1:L PR[91] R[100]mm/sec CNT100;
   1:  PR[91,1] = PR[90,1] + 5.063;
   1:  PR[91,2] = PR[90,2] + 30.322;
   1:L PR[91] R[100]mm/sec CNT100;
   1:  PR[91,1] = PR[90,1] + 5.074;
   1:  PR[91,2] = PR[90,2] + 30.294;
   1:L PR[91] R[100]mm/sec CNT100;
   1:  PR[91,1] = PR[90,1] + -0.738;
   1:  PR[91,2] = PR[90,2] + 24.482;
   1:L PR[91] R[100]mm/sec CNT100;
   1:  PR[91,2] = PR[90,2] + 20.240;
   1:L PR[91] R[100]mm/sec CNT100;
   1:  PR[91,1] = PR[90,1] + 6.946;
   1:  PR[91,2] = PR[90,2] + 27.923;
   1:L PR[91] R[100]mm/sec CNT100;
   1:  PR[91,1] = PR[90,1] + 7.573;
   1:  PR[91,2] = PR[90,2] + 27.417;
   1:L PR[91] R[100]mm/sec CNT100;
   1:  PR[91,1] = PR[90,1] + 9.083;
   1:  PR[91,2] = PR[90,2] + 27.019;
   1:L PR[91] R[100]mm/sec CNT100;
   1:  PR[91,1] = PR[90,1] + 9.949;
   1:  PR[91,2] = PR[90,2] + 26.921;
   1:L PR[91] R[100]mm/sec CNT100;
   1:  PR[91,1] = PR[90,1] + 10.173;
   1:  PR[91,2] = PR[90,2] + 26.908;
   1:L PR[91] R[100]mm/sec CNT100;
   1:  PR[91,1] = PR[90,1] + -0.737;
   1:  PR[91,2] = PR[90,2] + 15.997;
   1:L PR[91] R[100]mm/sec CNT100;
   1:  PR[91,2] = PR[90,2] + 11.755;
   1:L PR[91] R[100]mm/sec CNT100;
   1:  PR[91,1] = PR[90,1] + 4.959;
   1:  PR[91,2] = PR[90,2] + 17.450;
   1:L PR[91] R[100]mm/sec CNT100;
   1:  PR[91,1] = PR[90,1] + 4.837;
   1:  PR[91,2] = PR[90,2] + 16.945;
   1:L PR[91] R[100]mm/sec CNT100;
   1:  PR[91,1] = PR[90,1] + 4.664;
   1:  PR[91,2] = PR[90,2] + 15.574;
   1:L PR[91] R[100]mm/sec CNT100;
   1:  PR[91,1] = PR[90,1] + 4.665;
   1:  PR[91,2] = PR[90,2] + 12.914;
   1:L PR[91] R[100]mm/sec CNT100;
   1:  PR[91,1] = PR[90,1] + -0.737;
   1:  PR[91,2] = PR[90,2] + 7.513;
   1:L PR[91] R[100]mm/sec CNT100;
   1:  PR[91,1] = PR[90,1] + -0.736;
   1:  PR[91,2] = PR[90,2] + 3.270;
   1:L PR[91] R[100]mm/sec CNT100;
   1:  PR[91,1] = PR[90,1] + 4.666;
   1:  PR[91,2] = PR[90,2] + 8.672;
   1:L PR[91] R[100]mm/sec CNT100;
   1:  PR[91,1] = PR[90,1] + 4.667;
   1:  PR[91,2] = PR[90,2] + 4.431;
   1:L PR[91] R[100]mm/sec CNT100;
   1:  PR[91,1] = PR[90,1] + -0.588;
   1:  PR[91,2] = PR[90,2] + -0.824;
   1:L PR[91] R[100]mm/sec CNT100;
   1:  PR[91,1] = PR[90,1] + -0.495;
   1:  PR[91,2] = PR[90,2] + -1.359;
   1:L PR[91] R[100]mm/sec CNT100;
   1:  PR[91,1] = PR[90,1] + -0.485;
   1:  PR[91,2] = PR[90,2] + -1.468;
   1:L PR[91] R[100]mm/sec CNT100;
   1:  PR[91,1] = PR[90,1] + -0.428;
   1:  PR[91,2] = PR[90,2] + -1.699;
   1:L PR[91] R[100]mm/sec CNT100;
   1:  PR[91,1] = PR[90,1] + -0.399;
   1:  PR[91,2] = PR[90,2] + -1.771;
   1:L PR[91] R[100]mm/sec CNT100;
   1:  PR[91,1] = PR[90,1] + -0.040;
   1:  PR[91,2] = PR[90,2] + -3.031;
   1:L PR[91] R[100]mm/sec CNT100;
   1:  PR[91,1] = PR[90,1] + -0.022;
   1:  PR[91,2] = PR[90,2] + -3.318;
   1:L PR[91] R[100]mm/sec CNT100;
   1:  PR[91,1] = PR[90,1] + 0.095;
   1:  PR[91,2] = PR[90,2] + -3.827;
   1:L PR[91] R[100]mm/sec CNT100;
   1:  PR[91,1] = PR[90,1] + 0.164;
   1:  PR[91,2] = PR[90,2] + -4.315;
   1:L PR[91] R[100]mm/sec CNT100;
   1:  PR[91,1] = PR[90,1] + 4.824;
   1:  PR[91,2] = PR[90,2] + 0.345;
   1:L PR[91] R[100]mm/sec CNT100;
   1:  PR[91,1] = PR[90,1] + 4.928;
   1:  PR[91,2] = PR[90,2] + -0.199;
   1:L PR[91] R[100]mm/sec CNT100;
   1:  PR[91,1] = PR[90,1] + 4.943;
   1:  PR[91,2] = PR[90,2] + -0.523;
   1:L PR[91] R[100]mm/sec CNT100;
   1:  PR[91,1] = PR[90,1] + 5.148;
   1:  PR[91,2] = PR[90,2] + -1.228;
   1:L PR[91] R[100]mm/sec CNT100;
   1:  PR[91,1] = PR[90,1] + 5.173;
   1:  PR[91,2] = PR[90,2] + -1.625;
   1:L PR[91] R[100]mm/sec CNT100;
   1:  PR[91,1] = PR[90,1] + 5.351;
   1:  PR[91,2] = PR[90,2] + -2.178;
   1:L PR[91] R[100]mm/sec CNT100;
   1:  PR[91,1] = PR[90,1] + 5.381;
   1:  PR[91,2] = PR[90,2] + -2.508;
   1:L PR[91] R[100]mm/sec CNT100;
   1:  PR[91,1] = PR[90,1] + 5.533;
   1:  PR[91,2] = PR[90,2] + -3.189;
   1:L PR[91] R[100]mm/sec CNT100;
   1:  PR[91,1] = PR[90,1] + 1.308;
   1:  PR[91,2] = PR[90,2] + -7.413;
   1:L PR[91] R[100]mm/sec CNT100;
   1:  PR[91,1] = PR[90,1] + 1.818;
   1:  PR[91,2] = PR[90,2] + -8.056;
   1:L PR[91] R[100]mm/sec CNT100;
   1:  PR[91,1] = PR[90,1] + 1.968;
   1:  PR[91,2] = PR[90,2] + -8.964;
   1:L PR[91] R[100]mm/sec CNT100;
   1:  PR[91,1] = PR[90,1] + 1.970;
   1:  PR[91,2] = PR[90,2] + -8.969;
   1:L PR[91] R[100]mm/sec CNT100;
   1:  PR[91,1] = PR[90,1] + 2.724;
   1:  PR[91,2] = PR[90,2] + -9.748;
   1:L PR[91] R[100]mm/sec CNT100;
   1:  PR[91,1] = PR[90,1] + 2.815;
   1:  PR[91,2] = PR[90,2] + -10.149;
   1:L PR[91] R[100]mm/sec CNT100;
   1:  PR[91,1] = PR[90,1] + 6.749;
   1:  PR[91,2] = PR[90,2] + -6.215;
   1:L PR[91] R[100]mm/sec CNT100;
   1:  PR[91,1] = PR[90,1] + 7.037;
   1:  PR[91,2] = PR[90,2] + -7.202;
   1:L PR[91] R[100]mm/sec CNT100;
   1:  PR[91,1] = PR[90,1] + 7.801;
   1:  PR[91,2] = PR[90,2] + -7.993;
   1:L PR[91] R[100]mm/sec CNT100;
   1:  PR[91,1] = PR[90,1] + 8.080;
   1:  PR[91,2] = PR[90,2] + -8.470;
   1:L PR[91] R[100]mm/sec CNT100;
   1:  PR[91,1] = PR[90,1] + 8.263;
   1:  PR[91,2] = PR[90,2] + -8.731;
   1:L PR[91] R[100]mm/sec CNT100;
   1:  PR[91,1] = PR[90,1] + 8.307;
   1:  PR[91,2] = PR[90,2] + -8.900;
   1:L PR[91] R[100]mm/sec CNT100;
   1:  PR[91,1] = PR[90,1] + 4.581;
   1:  PR[91,2] = PR[90,2] + -12.626;
   1:L PR[91] R[100]mm/sec CNT100;
   1:  PR[91,1] = PR[90,1] + 4.619;
   1:  PR[91,2] = PR[90,2] + -12.748;
   1:L PR[91] R[100]mm/sec CNT100;
   1:  PR[91,1] = PR[90,1] + 5.271;
   1:  PR[91,2] = PR[90,2] + -13.048;
   1:L PR[91] R[100]mm/sec CNT100;
   1:  PR[91,1] = PR[90,1] + 5.576;
   1:  PR[91,2] = PR[90,2] + -14.118;
   1:L PR[91] R[100]mm/sec CNT100;
   1:  PR[91,1] = PR[90,1] + 5.730;
   1:  PR[91,2] = PR[90,2] + -14.261;
   1:L PR[91] R[100]mm/sec CNT100;
   1:  PR[91,1] = PR[90,1] + 5.968;
   1:  PR[91,2] = PR[90,2] + -14.547;
   1:L PR[91] R[100]mm/sec CNT100;
   1:  PR[91,1] = PR[90,1] + 6.057;
   1:  PR[91,2] = PR[90,2] + -14.575;
   1:L PR[91] R[100]mm/sec CNT100;
   1:  PR[91,1] = PR[90,1] + 6.447;
   1:  PR[91,2] = PR[90,2] + -15.002;
   1:L PR[91] R[100]mm/sec CNT100;
   1:  PR[91,1] = PR[90,1] + 10.284;
   1:  PR[91,2] = PR[90,2] + -11.166;
   1:L PR[91] R[100]mm/sec CNT100;
   1:  PR[91,1] = PR[90,1] + 10.619;
   1:  PR[91,2] = PR[90,2] + -11.389;
   1:L PR[91] R[100]mm/sec CNT100;
   1:  PR[91,1] = PR[90,1] + 11.062;
   1:  PR[91,2] = PR[90,2] + -11.963;
   1:L PR[91] R[100]mm/sec CNT100;
   1:  PR[91,1] = PR[90,1] + 12.058;
   1:  PR[91,2] = PR[90,2] + -12.626;
   1:L PR[91] R[100]mm/sec CNT100;
   1:  PR[91,1] = PR[90,1] + 12.578;
   1:  PR[91,2] = PR[90,2] + -13.048;
   1:L PR[91] R[100]mm/sec CNT100;
   1:  PR[91,1] = PR[90,1] + 12.614;
   1:  PR[91,2] = PR[90,2] + -13.078;
   1:L PR[91] R[100]mm/sec CNT100;
   1:  PR[91,1] = PR[90,1] + 8.880;
   1:  PR[91,2] = PR[90,2] + -16.812;
   1:L PR[91] R[100]mm/sec CNT100;
   1:  PR[91,1] = PR[90,1] + 9.118;
   1:  PR[91,2] = PR[90,2] + -17.249;
   1:L PR[91] R[100]mm/sec CNT100;
   1:  PR[91,1] = PR[90,1] + 9.472;
   1:  PR[91,2] = PR[90,2] + -17.390;
   1:L PR[91] R[100]mm/sec CNT100;
   1:  PR[91,1] = PR[90,1] + 10.115;
   1:  PR[91,2] = PR[90,2] + -18.095;
   1:L PR[91] R[100]mm/sec CNT100;
   1:  PR[91,1] = PR[90,1] + 10.274;
   1:  PR[91,2] = PR[90,2] + -18.186;
   1:L PR[91] R[100]mm/sec CNT100;
   1:  PR[91,1] = PR[90,1] + 11.260;
   1:  PR[91,2] = PR[90,2] + -18.387;
   1:L PR[91] R[100]mm/sec CNT100;
   1:  PR[91,1] = PR[90,1] + 11.381;
   1:  PR[91,2] = PR[90,2] + -18.554;
   1:L PR[91] R[100]mm/sec CNT100;
   1:  PR[91,1] = PR[90,1] + 15.229;
   1:  PR[91,2] = PR[90,2] + -14.706;
   1:L PR[91] R[100]mm/sec CNT100;
   1:  PR[91,1] = PR[90,1] + 16.099;
   1:  PR[91,2] = PR[90,2] + -15.118;
   1:L PR[91] R[100]mm/sec CNT100;
   1:  PR[91,1] = PR[90,1] + 16.989;
   1:  PR[91,2] = PR[90,2] + -15.377;
   1:L PR[91] R[100]mm/sec CNT100;
   1:  PR[91,1] = PR[90,1] + 17.084;
   1:  PR[91,2] = PR[90,2] + -15.392;
   1:L PR[91] R[100]mm/sec CNT100;
   1:  PR[91,1] = PR[90,1] + 17.652;
   1:  PR[91,2] = PR[90,2] + -15.688;
   1:L PR[91] R[100]mm/sec CNT100;
   1:  PR[91,1] = PR[90,1] + 17.783;
   1:  PR[91,2] = PR[90,2] + -15.705;
   1:L PR[91] R[100]mm/sec CNT100;
   1:  PR[91,1] = PR[90,1] + 18.261;
   1:  PR[91,2] = PR[90,2] + -15.916;
   1:L PR[91] R[100]mm/sec CNT100;
   1:  PR[91,1] = PR[90,1] + 14.028;
   1:  PR[91,2] = PR[90,2] + -20.150;
   1:L PR[91] R[100]mm/sec CNT100;
   1:  PR[91,1] = PR[90,1] + 14.412;
   1:  PR[91,2] = PR[90,2] + -20.205;
   1:L PR[91] R[100]mm/sec CNT100;
   1:  PR[91,1] = PR[90,1] + 15.152;
   1:  PR[91,2] = PR[90,2] + -20.709;
   1:L PR[91] R[100]mm/sec CNT100;
   1:  PR[91,1] = PR[90,1] + 15.389;
   1:  PR[91,2] = PR[90,2] + -20.793;
   1:L PR[91] R[100]mm/sec CNT100;
   1:  PR[91,1] = PR[90,1] + 15.531;
   1:  PR[91,2] = PR[90,2] + -20.823;
   1:L PR[91] R[100]mm/sec CNT100;
   1:  PR[91,1] = PR[90,1] + 16.112;
   1:  PR[91,2] = PR[90,2] + -20.897;
   1:L PR[91] R[100]mm/sec CNT100;
   1:  PR[91,1] = PR[90,1] + 17.145;
   1:  PR[91,2] = PR[90,2] + -21.275;
   1:L PR[91] R[100]mm/sec CNT100;
   1:  PR[91,1] = PR[90,1] + 21.911;
   1:  PR[91,2] = PR[90,2] + -16.509;
   1:L PR[91] R[100]mm/sec CNT100;
   1:  PR[91,1] = PR[90,1] + 22.182;
   1:  PR[91,2] = PR[90,2] + -16.517;
   1:L PR[91] R[100]mm/sec CNT100;
   1:  PR[91,1] = PR[90,1] + 22.663;
   1:  PR[91,2] = PR[90,2] + -16.560;
   1:L PR[91] R[100]mm/sec CNT100;
   1:  PR[91,1] = PR[90,1] + 23.201;
   1:  PR[91,2] = PR[90,2] + -16.574;
   1:L PR[91] R[100]mm/sec CNT100;
   1:  PR[91,1] = PR[90,1] + 23.786;
   1:  PR[91,2] = PR[90,2] + -16.609;
   1:L PR[91] R[100]mm/sec CNT100;
   1:  PR[91,1] = PR[90,1] + 23.807;
   1:  PR[91,2] = PR[90,2] + -16.614;
   1:L PR[91] R[100]mm/sec CNT100;
   1:  PR[91,1] = PR[90,1] + 24.621;
   1:  PR[91,2] = PR[90,2] + -17.003;
   1:L PR[91] R[100]mm/sec CNT100;
   1:  PR[91,1] = PR[90,1] + 24.791;
   1:  PR[91,2] = PR[90,2] + -17.029;
   1:L PR[91] R[100]mm/sec CNT100;
   1:  PR[91,1] = PR[90,1] + 24.801;
   1:  PR[91,2] = PR[90,2] + -17.033;
   1:L PR[91] R[100]mm/sec CNT100;
   1:  PR[91,1] = PR[90,1] + 25.174;
   1:  PR[91,2] = PR[90,2] + -17.488;
   1:L PR[91] R[100]mm/sec CNT100;
   1:  PR[91,1] = PR[90,1] + 20.727;
   1:  PR[91,2] = PR[90,2] + -21.935;
   1:L PR[91] R[100]mm/sec CNT100;
   1:  PR[92] = PR[91];
   1:  PR[92,3] = PR[92,3] + R[101];
   1:J PR[92] R[102]% CNT100;
   1:  PR[91,1] = PR[90,1] + 21.441;
   1:  PR[91,2] = PR[90,2] + 21.205;
   1:  PR[92] = PR[91];
   1:  PR[92,3] = PR[92,3] + R[101];
   1:J PR[92] R[102]% CNT100;
   1:L PR[91] 100mm/sec CNT100 RampTo R[100];
   1:  PR[91,1] = PR[90,1] + 25.717;
   1:  PR[91,2] = PR[90,2] + 25.481;
   1:L PR[91] R[100]mm/sec CNT100;
   1:  PR[91,1] = PR[90,1] + 25.446;
   1:  PR[91,2] = PR[90,2] + 25.730;
   1:L PR[91] R[100]mm/sec CNT100;
   1:  PR[91,1] = PR[90,1] + 25.356;
   1:  PR[91,2] = PR[90,2] + 25.900;
   1:L PR[91] R[100]mm/sec CNT100;
   1:  PR[91,1] = PR[90,1] + 25.169;
   1:  PR[91,2] = PR[90,2] + 25.998;
   1:L PR[91] R[100]mm/sec CNT100;
   1:  PR[91,1] = PR[90,1] + 24.812;
   1:  PR[91,2] = PR[90,2] + 26.394;
   1:L PR[91] R[100]mm/sec CNT100;
   1:  PR[91,1] = PR[90,1] + 24.628;
   1:  PR[91,2] = PR[90,2] + 26.423;
   1:L PR[91] R[100]mm/sec CNT100;
   1:  PR[91,1] = PR[90,1] + 23.707;
   1:  PR[91,2] = PR[90,2] + 26.821;
   1:L PR[91] R[100]mm/sec CNT100;
   1:  PR[91,1] = PR[90,1] + 23.201;
   1:  PR[91,2] = PR[90,2] + 26.844;
   1:L PR[91] R[100]mm/sec CNT100;
   1:  PR[91,1] = PR[90,1] + 22.838;
   1:  PR[91,2] = PR[90,2] + 26.845;
   1:L PR[91] R[100]mm/sec CNT100;
   1:  PR[91,1] = PR[90,1] + 17.193;
   1:  PR[91,2] = PR[90,2] + 21.200;
   1:L PR[91] R[100]mm/sec CNT100;
   1:  PR[91,1] = PR[90,1] + 12.945;
   1:  PR[91,2] = PR[90,2] + 21.194;
   1:L PR[91] R[100]mm/sec CNT100;
   1:  PR[91,1] = PR[90,1] + 18.599;
   1:  PR[91,2] = PR[90,2] + 26.848;
   1:L PR[91] R[100]mm/sec CNT100;
   1:  PR[91,1] = PR[90,1] + 14.360;
   1:  PR[91,2] = PR[90,2] + 26.852;
   1:L PR[91] R[100]mm/sec CNT100;
   1:  PR[91,1] = PR[90,1] + 8.431;
   1:  PR[91,2] = PR[90,2] + 20.923;
   1:L PR[91] R[100]mm/sec CNT100;
   1:  PR[92] = PR[91];
   1:  PR[92,3] = PR[92,3] + R[101];
   1:J PR[92] R[102]% CNT100;
   1:  PR[91,1] = PR[90,1] + -45.999;
   1:  PR[91,2] = PR[90,2] + -10.151;
   1:  PR[92] = PR[91];
   1:  PR[92,3] = PR[92,3] + R[101];
   1:J PR[92] R[102]% CNT100;
   1:L PR[91] 100mm/sec CNT100 RampTo R[100];
   1:  PR[91,1] = PR[90,1] + -45.311;
   1:  PR[91,2] = PR[90,2] + -9.165;
   1:L PR[91] R[100]mm/sec CNT100;
   1:  PR[91,1] = PR[90,1] + -44.719;
   1:  PR[91,2] = PR[90,2] + -8.147;
   1:L PR[91] R[100]mm/sec CNT100;
   1:  PR[91,1] = PR[90,1] + -43.925;
   1:  PR[91,2] = PR[90,2] + -7.032;
   1:L PR[91] R[100]mm/sec CNT100;
   1:  PR[91,1] = PR[90,1] + -43.023;
   1:  PR[91,2] = PR[90,2] + -5.954;
   1:L PR[91] R[100]mm/sec CNT100;
   1:  PR[91,1] = PR[90,1] + -42.504;
   1:  PR[91,2] = PR[90,2] + -5.379;
   1:L PR[91] R[100]mm/sec CNT100;
   1:  PR[91,1] = PR[90,1] + -41.920;
   1:  PR[91,2] = PR[90,2] + -4.812;
   1:L PR[91] R[100]mm/sec CNT100;
   1:  PR[91,1] = PR[90,1] + -41.332;
   1:  PR[91,2] = PR[90,2] + -4.319;
   1:L PR[91] R[100]mm/sec CNT100;
   1:  PR[91,1] = PR[90,1] + -40.111;
   1:  PR[91,2] = PR[90,2] + -3.466;
   1:L PR[91] R[100]mm/sec CNT100;
   1:  PR[91,1] = PR[90,1] + -38.905;
   1:  PR[91,2] = PR[90,2] + -3.028;
   1:L PR[91] R[100]mm/sec CNT100;
   1:  PR[91,1] = PR[90,1] + -38.088;
   1:  PR[91,2] = PR[90,2] + -2.751;
   1:L PR[91] R[100]mm/sec CNT100;
   1:  PR[91,1] = PR[90,1] + -37.729;
   1:  PR[91,2] = PR[90,2] + -2.682;
   1:L PR[91] R[100]mm/sec CNT100;
   1:  PR[91,1] = PR[90,1] + -36.638;
   1:  PR[91,2] = PR[90,2] + -2.406;
   1:L PR[91] R[100]mm/sec CNT100;
   1:  PR[91,1] = PR[90,1] + -35.397;
   1:  PR[91,2] = PR[90,2] + -2.318;
   1:L PR[91] R[100]mm/sec CNT100;
   1:  PR[91,1] = PR[90,1] + -34.103;
   1:  PR[91,2] = PR[90,2] + -2.404;
   1:L PR[91] R[100]mm/sec CNT100;
   1:  PR[91,1] = PR[90,1] + -33.321;
   1:  PR[91,2] = PR[90,2] + -2.642;
   1:L PR[91] R[100]mm/sec CNT100;
   1:  PR[91,1] = PR[90,1] + -33.036;
   1:  PR[91,2] = PR[90,2] + -2.665;
   1:L PR[91] R[100]mm/sec CNT100;
   1:  PR[91,1] = PR[90,1] + -32.433;
   1:  PR[91,2] = PR[90,2] + -2.906;
   1:L PR[91] R[100]mm/sec CNT100;
   1:  PR[91,1] = PR[90,1] + -32.041;
   1:  PR[91,2] = PR[90,2] + -2.968;
   1:L PR[91] R[100]mm/sec CNT100;
   1:  PR[91,1] = PR[90,1] + -31.495;
   1:  PR[91,2] = PR[90,2] + -3.134;
   1:L PR[91] R[100]mm/sec CNT100;
   1:  PR[91,1] = PR[90,1] + -30.951;
   1:  PR[91,2] = PR[90,2] + -3.369;
   1:L PR[91] R[100]mm/sec CNT100;
   1:  PR[91,1] = PR[90,1] + -30.436;
   1:  PR[91,2] = PR[90,2] + -3.452;
   1:L PR[91] R[100]mm/sec CNT100;
   1:  PR[91,1] = PR[90,1] + -30.094;
   1:  PR[91,2] = PR[90,2] + -3.931;
   1:L PR[91] R[100]mm/sec CNT100;
   1:  PR[91,1] = PR[90,1] + -29.970;
   1:  PR[91,2] = PR[90,2] + -4.050;
   1:L PR[91] R[100]mm/sec CNT100;
   1:  PR[91,1] = PR[90,1] + -29.166;
   1:  PR[91,2] = PR[90,2] + -4.359;
   1:L PR[91] R[100]mm/sec CNT100;
   1:  PR[91,1] = PR[90,1] + -28.644;
   1:  PR[91,2] = PR[90,2] + -4.979;
   1:L PR[91] R[100]mm/sec CNT100;
   1:  PR[91,1] = PR[90,1] + -28.128;
   1:  PR[91,2] = PR[90,2] + -5.298;
   1:L PR[91] R[100]mm/sec CNT100;
   1:  PR[91,1] = PR[90,1] + -27.718;
   1:  PR[91,2] = PR[90,2] + -5.601;
   1:L PR[91] R[100]mm/sec CNT100;
   1:  PR[91,1] = PR[90,1] + -27.690;
   1:  PR[91,2] = PR[90,2] + -5.607;
   1:L PR[91] R[100]mm/sec CNT100;
   1:  PR[91,1] = PR[90,1] + -27.492;
   1:  PR[91,2] = PR[90,2] + -5.769;
   1:L PR[91] R[100]mm/sec CNT100;
   1:  PR[91,1] = PR[90,1] + -27.269;
   1:  PR[91,2] = PR[90,2] + -5.934;
   1:L PR[91] R[100]mm/sec CNT100;
   1:  PR[91,1] = PR[90,1] + -27.253;
   1:  PR[91,2] = PR[90,2] + -5.964;
   1:L PR[91] R[100]mm/sec CNT100;
   1:  PR[91,1] = PR[90,1] + -27.111;
   1:  PR[91,2] = PR[90,2] + -6.080;
   1:L PR[91] R[100]mm/sec CNT100;
   1:  PR[91,1] = PR[90,1] + -26.954;
   1:  PR[91,2] = PR[90,2] + -6.129;
   1:L PR[91] R[100]mm/sec CNT100;
   1:  PR[91,1] = PR[90,1] + -26.481;
   1:  PR[91,2] = PR[90,2] + -6.242;
   1:L PR[91] R[100]mm/sec CNT100;
   1:  PR[91,1] = PR[90,1] + -25.613;
   1:  PR[91,2] = PR[90,2] + -6.762;
   1:L PR[91] R[100]mm/sec CNT100;
   1:  PR[91,1] = PR[90,1] + -25.301;
   1:  PR[91,2] = PR[90,2] + -6.923;
   1:L PR[91] R[100]mm/sec CNT100;
   1:  PR[91,1] = PR[90,1] + -25.065;
   1:  PR[91,2] = PR[90,2] + -6.957;
   1:L PR[91] R[100]mm/sec CNT100;
   1:  PR[91,1] = PR[90,1] + -24.644;
   1:  PR[91,2] = PR[90,2] + -7.056;
   1:L PR[91] R[100]mm/sec CNT100;
   1:  PR[91,1] = PR[90,1] + -24.186;
   1:  PR[91,2] = PR[90,2] + -7.118;
   1:L PR[91] R[100]mm/sec CNT100;
   1:  PR[91,1] = PR[90,1] + -23.859;
   1:  PR[91,2] = PR[90,2] + -7.140;
   1:L PR[91] R[100]mm/sec CNT100;
   1:  PR[91,1] = PR[90,1] + -23.194;
   1:  PR[91,2] = PR[90,2] + -7.233;
   1:L PR[91] R[100]mm/sec CNT100;
   1:  PR[91,1] = PR[90,1] + -22.327;
   1:  PR[91,2] = PR[90,2] + -7.274;
   1:L PR[91] R[100]mm/sec CNT100;
   1:  PR[91,1] = PR[90,1] + -21.205;
   1:  PR[91,2] = PR[90,2] + -7.222;
   1:L PR[91] R[100]mm/sec CNT100;
   1:  PR[91,1] = PR[90,1] + -20.556;
   1:  PR[91,2] = PR[90,2] + -7.146;
   1:L PR[91] R[100]mm/sec CNT100;
   1:  PR[91,1] = PR[90,1] + -20.151;
   1:  PR[91,2] = PR[90,2] + -7.063;
   1:L PR[91] R[100]mm/sec CNT100;
   1:  PR[91,1] = PR[90,1] + -19.688;
   1:  PR[91,2] = PR[90,2] + -7.003;
   1:L PR[91] R[100]mm/sec CNT100;
   1:  PR[91,1] = PR[90,1] + -18.924;
   1:  PR[91,2] = PR[90,2] + -6.705;
   1:L PR[91] R[100]mm/sec CNT100;
   1:  PR[91,1] = PR[90,1] + -18.836;
   1:  PR[91,2] = PR[90,2] + -6.689;
   1:L PR[91] R[100]mm/sec CNT100;
   1:  PR[91,1] = PR[90,1] + -18.706;
   1:  PR[91,2] = PR[90,2] + -6.614;
   1:L PR[91] R[100]mm/sec CNT100;
   1:  PR[91,1] = PR[90,1] + -17.988;
   1:  PR[91,2] = PR[90,2] + -6.290;
   1:L PR[91] R[100]mm/sec CNT100;
   1:  PR[91,1] = PR[90,1] + -17.219;
   1:  PR[91,2] = PR[90,2] + -5.846;
   1:L PR[91] R[100]mm/sec CNT100;
   1:  PR[91,1] = PR[90,1] + -17.071;
   1:  PR[91,2] = PR[90,2] + -5.784;
   1:L PR[91] R[100]mm/sec CNT100;
   1:  PR[91,1] = PR[90,1] + -17.008;
   1:  PR[91,2] = PR[90,2] + -5.733;
   1:L PR[91] R[100]mm/sec CNT100;
   1:  PR[91,1] = PR[90,1] + -16.228;
   1:  PR[91,2] = PR[90,2] + -5.194;
   1:L PR[91] R[100]mm/sec CNT100;
   1:  PR[91,1] = PR[90,1] + -15.829;
   1:  PR[91,2] = PR[90,2] + -4.832;
   1:L PR[91] R[100]mm/sec CNT100;
   1:  PR[91,1] = PR[90,1] + -15.364;
   1:  PR[91,2] = PR[90,2] + -4.381;
   1:L PR[91] R[100]mm/sec CNT100;
   1:  PR[91,1] = PR[90,1] + -14.965;
   1:  PR[91,2] = PR[90,2] + -3.945;
   1:L PR[91] R[100]mm/sec CNT100;
   1:  PR[91,1] = PR[90,1] + -14.314;
   1:  PR[91,2] = PR[90,2] + -3.111;
   1:L PR[91] R[100]mm/sec CNT100;
   1:  PR[91,1] = PR[90,1] + -14.132;
   1:  PR[91,2] = PR[90,2] + -2.726;
   1:L PR[91] R[100]mm/sec CNT100;
   1:  PR[91,1] = PR[90,1] + -13.362;
   1:  PR[91,2] = PR[90,2] + -1.352;
   1:L PR[91] R[100]mm/sec CNT100;
   1:  PR[91,1] = PR[90,1] + -13.305;
   1:  PR[91,2] = PR[90,2] + -1.069;
   1:L PR[91] R[100]mm/sec CNT100;
   1:  PR[91,1] = PR[90,1] + -13.108;
   1:  PR[91,2] = PR[90,2] + -0.460;
   1:L PR[91] R[100]mm/sec CNT100;
   1:  PR[91,1] = PR[90,1] + -12.933;
   1:  PR[91,2] = PR[90,2] + 0.266;
   1:L PR[91] R[100]mm/sec CNT100;
   1:  PR[91,1] = PR[90,1] + -12.723;
   1:  PR[91,2] = PR[90,2] + 1.365;
   1:L PR[91] R[100]mm/sec CNT100;
   1:  PR[91,1] = PR[90,1] + -12.647;
   1:  PR[91,2] = PR[90,2] + 2.202;
   1:L PR[91] R[100]mm/sec CNT100;
   1:  PR[91,1] = PR[90,1] + -12.685;
   1:  PR[91,2] = PR[90,2] + 3.038;
   1:L PR[91] R[100]mm/sec CNT100;
   1:  PR[91,1] = PR[90,1] + -12.744;
   1:  PR[91,2] = PR[90,2] + 3.270;
   1:L PR[91] R[100]mm/sec CNT100;
   1:  PR[91,1] = PR[90,1] + -12.842;
   1:  PR[91,2] = PR[90,2] + 3.896;
   1:L PR[91] R[100]mm/sec CNT100;
   1:  PR[91,1] = PR[90,1] + -13.030;
   1:  PR[91,2] = PR[90,2] + 4.664;
   1:L PR[91] R[100]mm/sec CNT100;
   1:  PR[91,1] = PR[90,1] + -13.064;
   1:  PR[91,2] = PR[90,2] + 4.984;
   1:L PR[91] R[100]mm/sec CNT100;
   1:  PR[91,1] = PR[90,1] + -13.149;
   1:  PR[91,2] = PR[90,2] + 5.440;
   1:L PR[91] R[100]mm/sec CNT100;
   1:  PR[91,1] = PR[90,1] + -13.289;
   1:  PR[91,2] = PR[90,2] + 5.905;
   1:L PR[91] R[100]mm/sec CNT100;
   1:  PR[91,1] = PR[90,1] + -13.303;
   1:  PR[91,2] = PR[90,2] + 6.022;
   1:L PR[91] R[100]mm/sec CNT100;
   1:  PR[91,1] = PR[90,1] + -13.595;
   1:  PR[91,2] = PR[90,2] + 6.383;
   1:L PR[91] R[100]mm/sec CNT100;
   1:  PR[91,1] = PR[90,1] + -14.209;
   1:  PR[91,2] = PR[90,2] + 7.676;
   1:L PR[91] R[100]mm/sec CNT100;
   1:  PR[91,1] = PR[90,1] + -14.744;
   1:  PR[91,2] = PR[90,2] + 8.156;
   1:L PR[91] R[100]mm/sec CNT100;
   1:  PR[91,1] = PR[90,1] + -14.978;
   1:  PR[91,2] = PR[90,2] + 8.726;
   1:L PR[91] R[100]mm/sec CNT100;
   1:  PR[91,1] = PR[90,1] + -15.519;
   1:  PR[91,2] = PR[90,2] + 9.047;
   1:L PR[91] R[100]mm/sec CNT100;
   1:  PR[91,1] = PR[90,1] + -15.841;
   1:  PR[91,2] = PR[90,2] + 9.611;
   1:L PR[91] R[100]mm/sec CNT100;
   1:  PR[91,1] = PR[90,1] + -16.428;
   1:  PR[91,2] = PR[90,2] + 9.876;
   1:L PR[91] R[100]mm/sec CNT100;
   1:  PR[91,1] = PR[90,1] + -16.833;
   1:  PR[91,2] = PR[90,2] + 10.394;
   1:L PR[91] R[100]mm/sec CNT100;
   1:  PR[91,1] = PR[90,1] + -17.335;
   1:  PR[91,2] = PR[90,2] + 10.617;
   1:L PR[91] R[100]mm/sec CNT100;
   1:  PR[91,1] = PR[90,1] + -17.867;
   1:  PR[91,2] = PR[90,2] + 10.946;
   1:L PR[91] R[100]mm/sec CNT100;
   1:  PR[91,1] = PR[90,1] + -17.888;
   1:  PR[91,2] = PR[90,2] + 10.949;
   1:L PR[91] R[100]mm/sec CNT100;
   1:  PR[91,1] = PR[90,1] + -17.984;
   1:  PR[91,2] = PR[90,2] + 11.017;
   1:L PR[91] R[100]mm/sec CNT100;
   1:  PR[91,1] = PR[90,1] + -18.295;
   1:  PR[91,2] = PR[90,2] + 11.210;
   1:L PR[91] R[100]mm/sec CNT100;
   1:  PR[91,1] = PR[90,1] + -18.325;
   1:  PR[91,2] = PR[90,2] + 11.262;
   1:L PR[91] R[100]mm/sec CNT100;
   1:  PR[91,1] = PR[90,1] + -18.422;
   1:  PR[91,2] = PR[90,2] + 11.332;
   1:L PR[91] R[100]mm/sec CNT100;
   1:  PR[91,1] = PR[90,1] + -18.619;
   1:  PR[91,2] = PR[90,2] + 11.363;
   1:L PR[91] R[100]mm/sec CNT100;
   1:  PR[91,1] = PR[90,1] + -19.589;
   1:  PR[91,2] = PR[90,2] + 11.623;
   1:L PR[91] R[100]mm/sec CNT100;
   1:  PR[91,1] = PR[90,1] + -19.796;
   1:  PR[91,2] = PR[90,2] + 11.645;
   1:L PR[91] R[100]mm/sec CNT100;
   1:  PR[91,1] = PR[90,1] + -20.617;
   1:  PR[91,2] = PR[90,2] + 11.904;
   1:L PR[91] R[100]mm/sec CNT100;
   1:  PR[91,1] = PR[90,1] + -20.698;
   1:  PR[91,2] = PR[90,2] + 11.946;
   1:L PR[91] R[100]mm/sec CNT100;
   1:  PR[91,1] = PR[90,1] + -21.255;
   1:  PR[91,2] = PR[90,2] + 12.071;
   1:L PR[91] R[100]mm/sec CNT100;
   1:  PR[91,1] = PR[90,1] + -22.319;
   1:  PR[91,2] = PR[90,2] + 12.117;
   1:L PR[91] R[100]mm/sec CNT100;
   1:  PR[91,1] = PR[90,1] + -23.148;
   1:  PR[91,2] = PR[90,2] + 12.071;
   1:L PR[91] R[100]mm/sec CNT100;
   1:  PR[91,1] = PR[90,1] + -23.916;
   1:  PR[91,2] = PR[90,2] + 11.921;
   1:L PR[91] R[100]mm/sec CNT100;
   1:  PR[91,1] = PR[90,1] + -24.044;
   1:  PR[91,2] = PR[90,2] + 11.871;
   1:L PR[91] R[100]mm/sec CNT100;
   1:  PR[91,1] = PR[90,1] + -25.820;
   1:  PR[91,2] = PR[90,2] + 11.381;
   1:L PR[91] R[100]mm/sec CNT100;
   1:  PR[91,1] = PR[90,1] + -26.665;
   1:  PR[91,2] = PR[90,2] + 10.975;
   1:L PR[91] R[100]mm/sec CNT100;
   1:  PR[91,1] = PR[90,1] + -27.536;
   1:  PR[91,2] = PR[90,2] + 10.493;
   1:L PR[91] R[100]mm/sec CNT100;
   1:  PR[91,1] = PR[90,1] + -28.061;
   1:  PR[91,2] = PR[90,2] + 10.093;
   1:L PR[91] R[100]mm/sec CNT100;
   1:  PR[91,1] = PR[90,1] + -29.536;
   1:  PR[91,2] = PR[90,2] + 8.900;
   1:L PR[91] R[100]mm/sec CNT100;
   1:  PR[91,1] = PR[90,1] + -30.640;
   1:  PR[91,2] = PR[90,2] + 8.310;
   1:L PR[91] R[100]mm/sec CNT100;
   1:  PR[91,1] = PR[90,1] + -31.283;
   1:  PR[91,2] = PR[90,2] + 7.932;
   1:L PR[91] R[100]mm/sec CNT100;
   1:  PR[91,1] = PR[90,1] + -31.882;
   1:  PR[91,2] = PR[90,2] + 7.629;
   1:L PR[91] R[100]mm/sec CNT100;
   1:  PR[91,1] = PR[90,1] + -32.274;
   1:  PR[91,2] = PR[90,2] + 7.550;
   1:L PR[91] R[100]mm/sec CNT100;
   1:  PR[91,1] = PR[90,1] + -33.065;
   1:  PR[91,2] = PR[90,2] + 7.339;
   1:L PR[91] R[100]mm/sec CNT100;
   1:  PR[91,1] = PR[90,1] + -33.731;
   1:  PR[91,2] = PR[90,2] + 7.227;
   1:L PR[91] R[100]mm/sec CNT100;
   1:  PR[91,1] = PR[90,1] + -34.929;
   1:  PR[91,2] = PR[90,2] + 7.138;
   1:L PR[91] R[100]mm/sec CNT100;
   1:  PR[91,1] = PR[90,1] + -35.432;
   1:  PR[91,2] = PR[90,2] + 7.130;
   1:L PR[91] R[100]mm/sec CNT100;
   1:  PR[91,1] = PR[90,1] + -36.038;
   1:  PR[91,2] = PR[90,2] + 7.170;
   1:L PR[91] R[100]mm/sec CNT100;
   1:  PR[91,1] = PR[90,1] + -36.563;
   1:  PR[91,2] = PR[90,2] + 7.183;
   1:L PR[91] R[100]mm/sec CNT100;
   1:  PR[91,1] = PR[90,1] + -37.072;
   1:  PR[91,2] = PR[90,2] + 7.283;
   1:L PR[91] R[100]mm/sec CNT100;
   1:  PR[91,1] = PR[90,1] + -37.606;
   1:  PR[91,2] = PR[90,2] + 7.322;
   1:L PR[91] R[100]mm/sec CNT100;
   1:  PR[91,1] = PR[90,1] + -38.108;
   1:  PR[91,2] = PR[90,2] + 7.423;
   1:L PR[91] R[100]mm/sec CNT100;
   1:  PR[91,1] = PR[90,1] + -38.738;
   1:  PR[91,2] = PR[90,2] + 7.592;
   1:L PR[91] R[100]mm/sec CNT100;
   1:  PR[91,1] = PR[90,1] + -39.164;
   1:  PR[91,2] = PR[90,2] + 7.670;
   1:L PR[91] R[100]mm/sec CNT100;
   1:  PR[91,1] = PR[90,1] + -39.773;
   1:  PR[91,2] = PR[90,2] + 8.098;
   1:L PR[91] R[100]mm/sec CNT100;
   1:  PR[91,1] = PR[90,1] + -39.843;
   1:  PR[91,2] = PR[90,2] + 8.169;
   1:L PR[91] R[100]mm/sec CNT100;
   1:  PR[91,1] = PR[90,1] + -39.956;
   1:  PR[91,2] = PR[90,2] + 8.190;
   1:L PR[91] R[100]mm/sec CNT100;
   1:  PR[91,1] = PR[90,1] + -40.516;
   1:  PR[91,2] = PR[90,2] + 8.527;
   1:L PR[91] R[100]mm/sec CNT100;
   1:  PR[91,1] = PR[90,1] + -40.960;
   1:  PR[91,2] = PR[90,2] + 8.730;
   1:L PR[91] R[100]mm/sec CNT100;
   1:  PR[91,1] = PR[90,1] + -41.474;
   1:  PR[91,2] = PR[90,2] + 8.893;
   1:L PR[91] R[100]mm/sec CNT100;
   1:  PR[91,1] = PR[90,1] + -41.942;
   1:  PR[91,2] = PR[90,2] + 9.598;
   1:L PR[91] R[100]mm/sec CNT100;
   1:  PR[91,1] = PR[90,1] + -42.745;
   1:  PR[91,2] = PR[90,2] + 9.988;
   1:L PR[91] R[100]mm/sec CNT100;
   1:  PR[91,1] = PR[90,1] + -43.109;
   1:  PR[91,2] = PR[90,2] + 10.809;
   1:L PR[91] R[100]mm/sec CNT100;
   1:  PR[91,1] = PR[90,1] + -43.779;
   1:  PR[91,2] = PR[90,2] + 11.278;
   1:L PR[91] R[100]mm/sec CNT100;
   1:  PR[91,1] = PR[90,1] + -43.915;
   1:  PR[91,2] = PR[90,2] + 11.715;
   1:L PR[91] R[100]mm/sec CNT100;
   1:  PR[91,1] = PR[90,1] + -44.098;
   1:  PR[91,2] = PR[90,2] + 12.073;
   1:L PR[91] R[100]mm/sec CNT100;
   1:  PR[91,1] = PR[90,1] + -44.409;
   1:  PR[91,2] = PR[90,2] + 12.462;
   1:L PR[91] R[100]mm/sec CNT100;
   1:  PR[91,1] = PR[90,1] + -44.413;
   1:  PR[91,2] = PR[90,2] + 12.464;
   1:L PR[91] R[100]mm/sec CNT100;
   1:  PR[91,1] = PR[90,1] + -45.036;
   1:  PR[91,2] = PR[90,2] + 13.252;
   1:L PR[91] R[100]mm/sec CNT100;
   1:  PR[91,1] = PR[90,1] + -45.277;
   1:  PR[91,2] = PR[90,2] + 13.849;
   1:L PR[91] R[100]mm/sec CNT100;
   1:  PR[91,1] = PR[90,1] + -45.313;
   1:  PR[91,2] = PR[90,2] + 14.000;
   1:L PR[91] R[100]mm/sec CNT100;
   1:  PR[91,1] = PR[90,1] + -45.709;
   1:  PR[91,2] = PR[90,2] + 14.369;
   1:L PR[91] R[100]mm/sec CNT100;
   1:  PR[91,1] = PR[90,1] + -46.139;
   1:  PR[91,2] = PR[90,2] + 15.255;
   1:L PR[91] R[100]mm/sec CNT100;
   1:  PR[91,1] = PR[90,1] + -46.397;
   1:  PR[91,2] = PR[90,2] + 15.706;
   1:L PR[91] R[100]mm/sec CNT100;
   1:  PR[91,1] = PR[90,1] + -46.947;
   1:  PR[91,2] = PR[90,2] + 16.249;
   1:L PR[91] R[100]mm/sec CNT100;
   1:  PR[91,1] = PR[90,1] + -47.184;
   1:  PR[91,2] = PR[90,2] + 16.814;
   1:L PR[91] R[100]mm/sec CNT100;
   1:  PR[91,1] = PR[90,1] + -47.212;
   1:  PR[91,2] = PR[90,2] + 16.900;
   1:L PR[91] R[100]mm/sec CNT100;
   1:  PR[91,1] = PR[90,1] + -47.783;
   1:  PR[91,2] = PR[90,2] + 17.296;
   1:L PR[91] R[100]mm/sec CNT100;
   1:  PR[91,1] = PR[90,1] + -47.949;
   1:  PR[91,2] = PR[90,2] + 17.739;
   1:L PR[91] R[100]mm/sec CNT100;
   1:  PR[91,1] = PR[90,1] + -48.074;
   1:  PR[91,2] = PR[90,2] + 17.976;
   1:L PR[91] R[100]mm/sec CNT100;
   1:  PR[91,1] = PR[90,1] + -48.237;
   1:  PR[91,2] = PR[90,2] + 18.116;
   1:L PR[91] R[100]mm/sec CNT100;
   1:  PR[91,1] = PR[90,1] + -48.386;
   1:  PR[91,2] = PR[90,2] + 18.167;
   1:L PR[91] R[100]mm/sec CNT100;
   1:  PR[91,1] = PR[90,1] + -48.534;
   1:  PR[91,2] = PR[90,2] + 18.369;
   1:L PR[91] R[100]mm/sec CNT100;
   1:  PR[91,1] = PR[90,1] + -48.717;
   1:  PR[91,2] = PR[90,2] + 18.524;
   1:L PR[91] R[100]mm/sec CNT100;
   1:  PR[91,1] = PR[90,1] + -48.757;
   1:  PR[91,2] = PR[90,2] + 18.672;
   1:L PR[91] R[100]mm/sec CNT100;
   1:  PR[91,1] = PR[90,1] + -48.980;
   1:  PR[91,2] = PR[90,2] + 18.975;
   1:L PR[91] R[100]mm/sec CNT100;
   1:  PR[91,1] = PR[90,1] + -49.262;
   1:  PR[91,2] = PR[90,2] + 19.239;
   1:L PR[91] R[100]mm/sec CNT100;
   1:  PR[91,1] = PR[90,1] + -49.309;
   1:  PR[91,2] = PR[90,2] + 19.254;
   1:L PR[91] R[100]mm/sec CNT100;
   1:  PR[91,1] = PR[90,1] + -49.455;
   1:  PR[91,2] = PR[90,2] + 19.420;
   1:L PR[91] R[100]mm/sec CNT100;
   1:  PR[91,1] = PR[90,1] + -49.611;
   1:  PR[91,2] = PR[90,2] + 19.565;
   1:L PR[91] R[100]mm/sec CNT100;
   1:  PR[91,1] = PR[90,1] + -49.624;
   1:  PR[91,2] = PR[90,2] + 19.611;
   1:L PR[91] R[100]mm/sec CNT100;
   1:  PR[91,1] = PR[90,1] + -49.916;
   1:  PR[91,2] = PR[90,2] + 19.942;
   1:L PR[91] R[100]mm/sec CNT100;
   1:  PR[91,1] = PR[90,1] + -50.240;
   1:  PR[91,2] = PR[90,2] + 20.234;
   1:L PR[91] R[100]mm/sec CNT100;
   1:  PR[91,1] = PR[90,1] + -50.281;
   1:  PR[91,2] = PR[90,2] + 20.246;
   1:L PR[91] R[100]mm/sec CNT100;
   1:  PR[91,1] = PR[90,1] + -50.425;
   1:  PR[91,2] = PR[90,2] + 20.401;
   1:L PR[91] R[100]mm/sec CNT100;
   1:  PR[91,1] = PR[90,1] + -50.591;
   1:  PR[91,2] = PR[90,2] + 20.550;
   1:L PR[91] R[100]mm/sec CNT100;
   1:  PR[91,1] = PR[90,1] + -50.604;
   1:  PR[91,2] = PR[90,2] + 20.593;
   1:L PR[91] R[100]mm/sec CNT100;
   1:  PR[91,1] = PR[90,1] + -50.880;
   1:  PR[91,2] = PR[90,2] + 20.890;
   1:L PR[91] R[100]mm/sec CNT100;
   1:  PR[91,1] = PR[90,1] + -51.191;
   1:  PR[91,2] = PR[90,2] + 21.132;
   1:L PR[91] R[100]mm/sec CNT100;
   1:  PR[91,1] = PR[90,1] + -51.305;
   1:  PR[91,2] = PR[90,2] + 21.164;
   1:L PR[91] R[100]mm/sec CNT100;
   1:  PR[91,1] = PR[90,1] + -51.461;
   1:  PR[91,2] = PR[90,2] + 21.343;
   1:L PR[91] R[100]mm/sec CNT100;
   1:  PR[91,1] = PR[90,1] + -51.658;
   1:  PR[91,2] = PR[90,2] + 21.496;
   1:L PR[91] R[100]mm/sec CNT100;
   1:  PR[91,1] = PR[90,1] + -51.697;
   1:  PR[91,2] = PR[90,2] + 21.614;
   1:L PR[91] R[100]mm/sec CNT100;
   1:  PR[91,1] = PR[90,1] + -51.871;
   1:  PR[91,2] = PR[90,2] + 21.813;
   1:L PR[91] R[100]mm/sec CNT100;
   1:  PR[91,1] = PR[90,1] + -52.132;
   1:  PR[91,2] = PR[90,2] + 21.969;
   1:L PR[91] R[100]mm/sec CNT100;
   1:  PR[91,1] = PR[90,1] + -52.495;
   1:  PR[91,2] = PR[90,2] + 22.110;
   1:L PR[91] R[100]mm/sec CNT100;
   1:  PR[91,1] = PR[90,1] + -52.929;
   1:  PR[91,2] = PR[90,2] + 22.710;
   1:L PR[91] R[100]mm/sec CNT100;
   1:  PR[91,1] = PR[90,1] + -53.609;
   1:  PR[91,2] = PR[90,2] + 22.992;
   1:L PR[91] R[100]mm/sec CNT100;
   1:  PR[91,1] = PR[90,1] + -54.054;
   1:  PR[91,2] = PR[90,2] + 23.557;
   1:L PR[91] R[100]mm/sec CNT100;
   1:  PR[91,1] = PR[90,1] + -54.631;
   1:  PR[91,2] = PR[90,2] + 23.854;
   1:L PR[91] R[100]mm/sec CNT100;
   1:  PR[91,1] = PR[90,1] + -55.406;
   1:  PR[91,2] = PR[90,2] + 24.488;
   1:L PR[91] R[100]mm/sec CNT100;
   1:  PR[91,1] = PR[90,1] + -55.408;
   1:  PR[91,2] = PR[90,2] + 24.492;
   1:L PR[91] R[100]mm/sec CNT100;
   1:  PR[91,1] = PR[90,1] + -55.678;
   1:  PR[91,2] = PR[90,2] + 24.701;
   1:L PR[91] R[100]mm/sec CNT100;
   1:  PR[91,1] = PR[90,1] + -55.998;
   1:  PR[91,2] = PR[90,2] + 24.832;
   1:L PR[91] R[100]mm/sec CNT100;
   1:  PR[91,1] = PR[90,1] + -56.456;
   1:  PR[91,2] = PR[90,2] + 24.972;
   1:L PR[91] R[100]mm/sec CNT100;
   1:  PR[91,1] = PR[90,1] + -56.931;
   1:  PR[91,2] = PR[90,2] + 25.462;
   1:L PR[91] R[100]mm/sec CNT100;
   1:  PR[91,1] = PR[90,1] + -56.946;
   1:  PR[91,2] = PR[90,2] + 25.481;
   1:L PR[91] R[100]mm/sec CNT100;
   1:  PR[91,1] = PR[90,1] + -56.977;
   1:  PR[91,2] = PR[90,2] + 25.487;
   1:L PR[91] R[100]mm/sec CNT100;
   1:  PR[91,1] = PR[90,1] + -58.393;
   1:  PR[91,2] = PR[90,2] + 26.167;
   1:L PR[91] R[100]mm/sec CNT100;
   1:  PR[91,1] = PR[90,1] + -58.764;
   1:  PR[91,2] = PR[90,2] + 26.509;
   1:L PR[91] R[100]mm/sec CNT100;
   1:  PR[91,1] = PR[90,1] + -58.896;
   1:  PR[91,2] = PR[90,2] + 26.533;
   1:L PR[91] R[100]mm/sec CNT100;
   1:  PR[91,1] = PR[90,1] + -59.420;
   1:  PR[91,2] = PR[90,2] + 26.717;
   1:L PR[91] R[100]mm/sec CNT100;
   1:  PR[91,1] = PR[90,1] + -59.972;
   1:  PR[91,2] = PR[90,2] + 26.963;
   1:L PR[91] R[100]mm/sec CNT100;
   1:  PR[91,1] = PR[90,1] + -60.227;
   1:  PR[91,2] = PR[90,2] + 27.014;
   1:L PR[91] R[100]mm/sec CNT100;
   1:  PR[91,1] = PR[90,1] + -60.751;
   1:  PR[91,2] = PR[90,2] + 27.436;
   1:L PR[91] R[100]mm/sec CNT100;
   1:  PR[91,1] = PR[90,1] + -60.891;
   1:  PR[91,2] = PR[90,2] + 27.456;
   1:L PR[91] R[100]mm/sec CNT100;
   1:  PR[91,1] = PR[90,1] + -61.377;
   1:  PR[91,2] = PR[90,2] + 27.636;
   1:L PR[91] R[100]mm/sec CNT100;
   1:  PR[91,1] = PR[90,1] + -61.839;
   1:  PR[91,2] = PR[90,2] + 27.754;
   1:L PR[91] R[100]mm/sec CNT100;
   1:  PR[91,1] = PR[90,1] + -62.201;
   1:  PR[91,2] = PR[90,2] + 27.817;
   1:L PR[91] R[100]mm/sec CNT100;
   1:  PR[91,1] = PR[90,1] + -63.042;
   1:  PR[91,2] = PR[90,2] + 28.213;
   1:L PR[91] R[100]mm/sec CNT100;
   1:  PR[91,1] = PR[90,1] + -63.078;
   1:  PR[91,2] = PR[90,2] + 28.244;
   1:L PR[91] R[100]mm/sec CNT100;
   1:  PR[91,1] = PR[90,1] + -63.516;
   1:  PR[91,2] = PR[90,2] + 28.455;
   1:L PR[91] R[100]mm/sec CNT100;
   1:  PR[91,1] = PR[90,1] + -63.797;
   1:  PR[91,2] = PR[90,2] + 28.485;
   1:L PR[91] R[100]mm/sec CNT100;
   1:  PR[91,1] = PR[90,1] + -64.238;
   1:  PR[91,2] = PR[90,2] + 28.596;
   1:L PR[91] R[100]mm/sec CNT100;
   1:  PR[91,1] = PR[90,1] + -65.116;
   1:  PR[91,2] = PR[90,2] + 28.713;
   1:L PR[91] R[100]mm/sec CNT100;
   1:  PR[91,1] = PR[90,1] + -65.775;
   1:  PR[91,2] = PR[90,2] + 28.871;
   1:L PR[91] R[100]mm/sec CNT100;
   1:  PR[91,1] = PR[90,1] + -65.911;
   1:  PR[91,2] = PR[90,2] + 28.881;
   1:L PR[91] R[100]mm/sec CNT100;
   1:  PR[91,1] = PR[90,1] + -66.626;
   1:  PR[91,2] = PR[90,2] + 29.060;
   1:L PR[91] R[100]mm/sec CNT100;
   1:  PR[91,1] = PR[90,1] + -66.783;
   1:  PR[91,2] = PR[90,2] + 29.119;
   1:L PR[91] R[100]mm/sec CNT100;
   1:  PR[91,1] = PR[90,1] + -67.483;
   1:  PR[91,2] = PR[90,2] + 29.270;
   1:L PR[91] R[100]mm/sec CNT100;
   1:  PR[91,1] = PR[90,1] + -67.679;
   1:  PR[91,2] = PR[90,2] + 29.279;
   1:L PR[91] R[100]mm/sec CNT100;
   1:  PR[91,1] = PR[90,1] + -68.321;
   1:  PR[91,2] = PR[90,2] + 29.356;
   1:L PR[91] R[100]mm/sec CNT100;
   1:  PR[91,1] = PR[90,1] + -69.197;
   1:  PR[91,2] = PR[90,2] + 29.389;
   1:L PR[91] R[100]mm/sec CNT100;
   1:  PR[91,1] = PR[90,1] + -70.517;
   1:  PR[91,2] = PR[90,2] + 29.383;
   1:L PR[91] R[100]mm/sec CNT100;
   1:  PR[91,1] = PR[90,1] + -71.168;
   1:  PR[91,2] = PR[90,2] + 29.340;
   1:L PR[91] R[100]mm/sec CNT100;
   1:  PR[91,1] = PR[90,1] + -71.470;
   1:  PR[91,2] = PR[90,2] + 29.334;
   1:L PR[91] R[100]mm/sec CNT100;
   1:  PR[91,1] = PR[90,1] + -72.218;
   1:  PR[91,2] = PR[90,2] + 29.244;
   1:L PR[91] R[100]mm/sec CNT100;
   1:  PR[91,1] = PR[90,1] + -72.418;
   1:  PR[91,2] = PR[90,2] + 29.237;
   1:L PR[91] R[100]mm/sec CNT100;
   1:  PR[91,1] = PR[90,1] + -73.241;
   1:  PR[91,2] = PR[90,2] + 29.087;
   1:L PR[91] R[100]mm/sec CNT100;
   1:  PR[91,1] = PR[90,1] + -73.413;
   1:  PR[91,2] = PR[90,2] + 29.037;
   1:L PR[91] R[100]mm/sec CNT100;
   1:  PR[91,1] = PR[90,1] + -74.355;
   1:  PR[91,2] = PR[90,2] + 28.843;
   1:L PR[91] R[100]mm/sec CNT100;
   1:  PR[91,1] = PR[90,1] + -74.542;
   1:  PR[91,2] = PR[90,2] + 28.822;
   1:L PR[91] R[100]mm/sec CNT100;
   1:  PR[91,1] = PR[90,1] + -75.781;
   1:  PR[91,2] = PR[90,2] + 28.565;
   1:L PR[91] R[100]mm/sec CNT100;
   1:  PR[91,1] = PR[90,1] + -76.252;
   1:  PR[91,2] = PR[90,2] + 28.496;
   1:L PR[91] R[100]mm/sec CNT100;
   1:  PR[91,1] = PR[90,1] + -77.057;
   1:  PR[91,2] = PR[90,2] + 28.230;
   1:L PR[91] R[100]mm/sec CNT100;
   1:  PR[91,1] = PR[90,1] + -77.165;
   1:  PR[91,2] = PR[90,2] + 28.216;
   1:L PR[91] R[100]mm/sec CNT100;
   1:  PR[91,1] = PR[90,1] + -77.379;
   1:  PR[91,2] = PR[90,2] + 28.110;
   1:L PR[91] R[100]mm/sec CNT100;
   1:  PR[91,1] = PR[90,1] + -78.121;
   1:  PR[91,2] = PR[90,2] + 27.820;
   1:L PR[91] R[100]mm/sec CNT100;
   1:  PR[91,1] = PR[90,1] + -79.059;
   1:  PR[91,2] = PR[90,2] + 27.539;
   1:L PR[91] R[100]mm/sec CNT100;
   1:  PR[91,1] = PR[90,1] + -79.979;
   1:  PR[91,2] = PR[90,2] + 27.078;
   1:L PR[91] R[100]mm/sec CNT100;
   1:  PR[91,1] = PR[90,1] + -80.953;
   1:  PR[91,2] = PR[90,2] + 26.646;
   1:L PR[91] R[100]mm/sec CNT100;
   1:  PR[91,1] = PR[90,1] + -82.086;
   1:  PR[91,2] = PR[90,2] + 26.012;
   1:L PR[91] R[100]mm/sec CNT100;
   1:  PR[91,1] = PR[90,1] + -83.481;
   1:  PR[91,2] = PR[90,2] + 25.528;
   1:L PR[91] R[100]mm/sec CNT100;
   1:  PR[91,1] = PR[90,1] + -84.987;
   1:  PR[91,2] = PR[90,2] + 25.731;
   1:L PR[91] R[100]mm/sec CNT100;
   1:  PR[91,1] = PR[90,1] + -85.524;
   1:  PR[91,2] = PR[90,2] + 26.856;
   1:L PR[91] R[100]mm/sec CNT100;
   1:  PR[91,1] = PR[90,1] + -85.760;
   1:  PR[91,2] = PR[90,2] + 27.443;
   1:L PR[91] R[100]mm/sec CNT100;
   1:  PR[91,1] = PR[90,1] + -85.889;
   1:  PR[91,2] = PR[90,2] + 28.633;
   1:L PR[91] R[100]mm/sec CNT100;
   1:  PR[91,1] = PR[90,1] + -85.909;
   1:  PR[91,2] = PR[90,2] + 30.486;
   1:L PR[91] R[100]mm/sec CNT100;
   1:  PR[91,1] = PR[90,1] + -85.910;
   1:  PR[91,2] = PR[90,2] + 40.599;
   1:L PR[91] R[100]mm/sec CNT100;
   1:  PR[91,1] = PR[90,1] + -85.928;
   1:  PR[91,2] = PR[90,2] + 41.736;
   1:L PR[91] R[100]mm/sec CNT100;
   1:  PR[91,1] = PR[90,1] + -85.997;
   1:  PR[91,2] = PR[90,2] + 42.330;
   1:L PR[91] R[100]mm/sec CNT100;
   1:  PR[91,1] = PR[90,1] + -86.050;
   1:  PR[91,2] = PR[90,2] + 42.444;
   1:L PR[91] R[100]mm/sec CNT100;
   1:  PR[91,1] = PR[90,1] + -86.271;
   1:  PR[91,2] = PR[90,2] + 43.211;
   1:L PR[91] R[100]mm/sec CNT100;
   1:  PR[91,1] = PR[90,1] + -86.284;
   1:  PR[91,2] = PR[90,2] + 43.350;
   1:L PR[91] R[100]mm/sec CNT100;
   1:  PR[91,1] = PR[90,1] + -86.578;
   1:  PR[91,2] = PR[90,2] + 44.309;
   1:L PR[91] R[100]mm/sec CNT100;
   1:  PR[91,1] = PR[90,1] + -86.585;
   1:  PR[91,2] = PR[90,2] + 44.350;
   1:L PR[91] R[100]mm/sec CNT100;
   1:  PR[91,1] = PR[90,1] + -87.016;
   1:  PR[91,2] = PR[90,2] + 44.743;
   1:L PR[91] R[100]mm/sec CNT100;
   1:  PR[91,1] = PR[90,1] + -87.125;
   1:  PR[91,2] = PR[90,2] + 45.061;
   1:L PR[91] R[100]mm/sec CNT100;
   1:  PR[91,1] = PR[90,1] + -87.259;
   1:  PR[91,2] = PR[90,2] + 45.305;
   1:L PR[91] R[100]mm/sec CNT100;
   1:  PR[91,1] = PR[90,1] + -87.392;
   1:  PR[91,2] = PR[90,2] + 45.423;
   1:L PR[91] R[100]mm/sec CNT100;
   1:  PR[91,1] = PR[90,1] + -87.452;
   1:  PR[91,2] = PR[90,2] + 45.439;
   1:L PR[91] R[100]mm/sec CNT100;
   1:  PR[91,1] = PR[90,1] + -87.646;
   1:  PR[91,2] = PR[90,2] + 45.648;
   1:L PR[91] R[100]mm/sec CNT100;
   1:  PR[91,1] = PR[90,1] + -87.876;
   1:  PR[91,2] = PR[90,2] + 45.852;
   1:L PR[91] R[100]mm/sec CNT100;
   1:  PR[91,1] = PR[90,1] + -87.893;
   1:  PR[91,2] = PR[90,2] + 45.915;
   1:L PR[91] R[100]mm/sec CNT100;
   1:  PR[91,1] = PR[90,1] + -87.997;
   1:  PR[91,2] = PR[90,2] + 46.026;
   1:L PR[91] R[100]mm/sec CNT100;
   1:  PR[91,1] = PR[90,1] + -88.215;
   1:  PR[91,2] = PR[90,2] + 46.132;
   1:L PR[91] R[100]mm/sec CNT100;
   1:  PR[91,1] = PR[90,1] + -88.560;
   1:  PR[91,2] = PR[90,2] + 46.243;
   1:L PR[91] R[100]mm/sec CNT100;
   1:  PR[91,1] = PR[90,1] + -88.980;
   1:  PR[91,2] = PR[90,2] + 46.638;
   1:L PR[91] R[100]mm/sec CNT100;
   1:  PR[91,1] = PR[90,1] + -89.017;
   1:  PR[91,2] = PR[90,2] + 46.678;
   1:L PR[91] R[100]mm/sec CNT100;
   1:  PR[91,1] = PR[90,1] + -89.468;
   1:  PR[91,2] = PR[90,2] + 46.826;
   1:L PR[91] R[100]mm/sec CNT100;
   1:  PR[91,1] = PR[90,1] + -89.879;
   1:  PR[91,2] = PR[90,2] + 46.909;
   1:L PR[91] R[100]mm/sec CNT100;
   1:  PR[91,1] = PR[90,1] + -90.142;
   1:  PR[91,2] = PR[90,2] + 46.932;
   1:L PR[91] R[100]mm/sec CNT100;
   1:  PR[91,1] = PR[90,1] + -90.809;
   1:  PR[91,2] = PR[90,2] + 47.050;
   1:L PR[91] R[100]mm/sec CNT100;
   1:  PR[91,1] = PR[90,1] + -91.579;
   1:  PR[91,2] = PR[90,2] + 47.057;
   1:L PR[91] R[100]mm/sec CNT100;
   1:  PR[91,1] = PR[90,1] + -92.406;
   1:  PR[91,2] = PR[90,2] + 46.942;
   1:L PR[91] R[100]mm/sec CNT100;
   1:  PR[91,1] = PR[90,1] + -93.150;
   1:  PR[91,2] = PR[90,2] + 46.769;
   1:L PR[91] R[100]mm/sec CNT100;
   1:  PR[91,1] = PR[90,1] + -93.816;
   1:  PR[91,2] = PR[90,2] + 46.411;
   1:L PR[91] R[100]mm/sec CNT100;
   1:  PR[91,1] = PR[90,1] + -94.745;
   1:  PR[91,2] = PR[90,2] + 45.772;
   1:L PR[91] R[100]mm/sec CNT100;
   1:  PR[91,1] = PR[90,1] + -94.858;
   1:  PR[91,2] = PR[90,2] + 45.664;
   1:L PR[91] R[100]mm/sec CNT100;
   1:  PR[91,1] = PR[90,1] + -95.468;
   1:  PR[91,2] = PR[90,2] + 44.911;
   1:L PR[91] R[100]mm/sec CNT100;
   1:  PR[91,1] = PR[90,1] + -95.478;
   1:  PR[91,2] = PR[90,2] + 44.884;
   1:L PR[91] R[100]mm/sec CNT100;
   1:  PR[91,1] = PR[90,1] + -95.973;
   1:  PR[91,2] = PR[90,2] + 44.032;
   1:L PR[91] R[100]mm/sec CNT100;
   1:  PR[91,1] = PR[90,1] + -96.252;
   1:  PR[91,2] = PR[90,2] + 43.218;
   1:L PR[91] R[100]mm/sec CNT100;
   1:  PR[91,1] = PR[90,1] + -96.487;
   1:  PR[91,2] = PR[90,2] + 42.400;
   1:L PR[91] R[100]mm/sec CNT100;
   1:  PR[91,1] = PR[90,1] + -96.492;
   1:  PR[91,2] = PR[90,2] + 42.252;
   1:L PR[91] R[100]mm/sec CNT100;
   1:  PR[91,1] = PR[90,1] + -96.561;
   1:  PR[91,2] = PR[90,2] + 41.543;
   1:L PR[91] R[100]mm/sec CNT100;
   1:  PR[91,1] = PR[90,1] + -96.570;
   1:  PR[91,2] = PR[90,2] + 40.604;
   1:L PR[91] R[100]mm/sec CNT100;
   1:  PR[91,1] = PR[90,1] + -96.569;
   1:  PR[91,2] = PR[90,2] + 3.184;
   1:L PR[91] R[100]mm/sec CNT100;
   1:  PR[91,1] = PR[90,1] + -96.559;
   1:  PR[91,2] = PR[90,2] + 1.842;
   1:L PR[91] R[100]mm/sec CNT100;
   1:  PR[91,1] = PR[90,1] + -96.528;
   1:  PR[91,2] = PR[90,2] + 0.910;
   1:L PR[91] R[100]mm/sec CNT100;
   1:  PR[91,1] = PR[90,1] + -96.467;
   1:  PR[91,2] = PR[90,2] + 0.033;
   1:L PR[91] R[100]mm/sec CNT100;
   1:  PR[91,1] = PR[90,1] + -96.367;
   1:  PR[91,2] = PR[90,2] + -0.755;
   1:L PR[91] R[100]mm/sec CNT100;
   1:  PR[91,1] = PR[90,1] + -96.238;
   1:  PR[91,2] = PR[90,2] + -1.347;
   1:L PR[91] R[100]mm/sec CNT100;
   1:  PR[91,1] = PR[90,1] + -96.003;
   1:  PR[91,2] = PR[90,2] + -2.491;
   1:L PR[91] R[100]mm/sec CNT100;
   1:  PR[91,1] = PR[90,1] + -95.992;
   1:  PR[91,2] = PR[90,2] + -2.712;
   1:L PR[91] R[100]mm/sec CNT100;
   1:  PR[91,1] = PR[90,1] + -95.875;
   1:  PR[91,2] = PR[90,2] + -3.325;
   1:L PR[91] R[100]mm/sec CNT100;
   1:  PR[91,1] = PR[90,1] + -95.773;
   1:  PR[91,2] = PR[90,2] + -4.186;
   1:L PR[91] R[100]mm/sec CNT100;
   1:  PR[91,1] = PR[90,1] + -95.660;
   1:  PR[91,2] = PR[90,2] + -4.638;
   1:L PR[91] R[100]mm/sec CNT100;
   1:  PR[91,1] = PR[90,1] + -95.625;
   1:  PR[91,2] = PR[90,2] + -4.917;
   1:L PR[91] R[100]mm/sec CNT100;
   1:  PR[91,1] = PR[90,1] + -95.408;
   1:  PR[91,2] = PR[90,2] + -5.439;
   1:L PR[91] R[100]mm/sec CNT100;
   1:  PR[91,1] = PR[90,1] + -95.396;
   1:  PR[91,2] = PR[90,2] + -5.456;
   1:L PR[91] R[100]mm/sec CNT100;
   1:  PR[91,1] = PR[90,1] + -95.002;
   1:  PR[91,2] = PR[90,2] + -6.288;
   1:L PR[91] R[100]mm/sec CNT100;
   1:  PR[91,1] = PR[90,1] + -94.962;
   1:  PR[91,2] = PR[90,2] + -6.651;
   1:L PR[91] R[100]mm/sec CNT100;
   1:  PR[91,1] = PR[90,1] + -94.691;
   1:  PR[91,2] = PR[90,2] + -7.613;
   1:L PR[91] R[100]mm/sec CNT100;
   1:  PR[91,1] = PR[90,1] + -94.661;
   1:  PR[91,2] = PR[90,2] + -7.783;
   1:L PR[91] R[100]mm/sec CNT100;
   1:  PR[91,1] = PR[90,1] + -94.392;
   1:  PR[91,2] = PR[90,2] + -8.202;
   1:L PR[91] R[100]mm/sec CNT100;
   1:  PR[91,1] = PR[90,1] + -93.932;
   1:  PR[91,2] = PR[90,2] + -9.081;
   1:L PR[91] R[100]mm/sec CNT100;
   1:  PR[91,1] = PR[90,1] + -93.753;
   1:  PR[91,2] = PR[90,2] + -9.790;
   1:L PR[91] R[100]mm/sec CNT100;
   1:  PR[91,1] = PR[90,1] + -93.614;
   1:  PR[91,2] = PR[90,2] + -9.989;
   1:L PR[91] R[100]mm/sec CNT100;
   1:  PR[91,1] = PR[90,1] + -93.593;
   1:  PR[91,2] = PR[90,2] + -10.004;
   1:L PR[91] R[100]mm/sec CNT100;
   1:  PR[91,1] = PR[90,1] + -93.463;
   1:  PR[91,2] = PR[90,2] + -10.203;
   1:L PR[91] R[100]mm/sec CNT100;
   1:  PR[91,1] = PR[90,1] + -93.324;
   1:  PR[91,2] = PR[90,2] + -10.402;
   1:L PR[91] R[100]mm/sec CNT100;
   1:  PR[91,1] = PR[90,1] + -93.320;
   1:  PR[91,2] = PR[90,2] + -10.424;
   1:L PR[91] R[100]mm/sec CNT100;
   1:  PR[91,1] = PR[90,1] + -92.965;
   1:  PR[91,2] = PR[90,2] + -10.972;
   1:L PR[91] R[100]mm/sec CNT100;
   1:  PR[91,1] = PR[90,1] + -92.768;
   1:  PR[91,2] = PR[90,2] + -11.555;
   1:L PR[91] R[100]mm/sec CNT100;
   1:  PR[91,1] = PR[90,1] + -92.752;
   1:  PR[91,2] = PR[90,2] + -11.613;
   1:L PR[91] R[100]mm/sec CNT100;
   1:  PR[91,1] = PR[90,1] + -92.723;
   1:  PR[91,2] = PR[90,2] + -11.642;
   1:L PR[91] R[100]mm/sec CNT100;
   1:  PR[91,1] = PR[90,1] + -92.216;
   1:  PR[91,2] = PR[90,2] + -11.998;
   1:L PR[91] R[100]mm/sec CNT100;
   1:  PR[91,1] = PR[90,1] + -92.113;
   1:  PR[91,2] = PR[90,2] + -12.491;
   1:L PR[91] R[100]mm/sec CNT100;
   1:  PR[91,1] = PR[90,1] + -91.948;
   1:  PR[91,2] = PR[90,2] + -12.801;
   1:L PR[91] R[100]mm/sec CNT100;
   1:  PR[91,1] = PR[90,1] + -91.643;
   1:  PR[91,2] = PR[90,2] + -13.262;
   1:L PR[91] R[100]mm/sec CNT100;
   1:  PR[91,1] = PR[90,1] + -91.078;
   1:  PR[91,2] = PR[90,2] + -13.818;
   1:L PR[91] R[100]mm/sec CNT100;
   1:  PR[91,1] = PR[90,1] + -90.816;
   1:  PR[91,2] = PR[90,2] + -14.416;
   1:L PR[91] R[100]mm/sec CNT100;
   1:  PR[91,1] = PR[90,1] + -90.198;
   1:  PR[91,2] = PR[90,2] + -14.812;
   1:L PR[91] R[100]mm/sec CNT100;
   1:  PR[91,1] = PR[90,1] + -89.967;
   1:  PR[91,2] = PR[90,2] + -15.448;
   1:L PR[91] R[100]mm/sec CNT100;
   1:  PR[91,1] = PR[90,1] + -89.948;
   1:  PR[91,2] = PR[90,2] + -15.486;
   1:L PR[91] R[100]mm/sec CNT100;
   1:  PR[91,1] = PR[90,1] + -89.922;
   1:  PR[91,2] = PR[90,2] + -15.504;
   1:L PR[91] R[100]mm/sec CNT100;
   1:  PR[91,1] = PR[90,1] + -89.305;
   1:  PR[91,2] = PR[90,2] + -15.784;
   1:L PR[91] R[100]mm/sec CNT100;
   1:  PR[91,1] = PR[90,1] + -89.085;
   1:  PR[91,2] = PR[90,2] + -16.400;
   1:L PR[91] R[100]mm/sec CNT100;
   1:  PR[91,1] = PR[90,1] + -89.036;
   1:  PR[91,2] = PR[90,2] + -16.478;
   1:L PR[91] R[100]mm/sec CNT100;
   1:  PR[91,1] = PR[90,1] + -88.963;
   1:  PR[91,2] = PR[90,2] + -16.529;
   1:L PR[91] R[100]mm/sec CNT100;
   1:  PR[91,1] = PR[90,1] + -88.365;
   1:  PR[91,2] = PR[90,2] + -16.758;
   1:L PR[91] R[100]mm/sec CNT100;
   1:  PR[91,1] = PR[90,1] + -88.130;
   1:  PR[91,2] = PR[90,2] + -17.359;
   1:L PR[91] R[100]mm/sec CNT100;
   1:  PR[91,1] = PR[90,1] + -88.082;
   1:  PR[91,2] = PR[90,2] + -17.429;
   1:L PR[91] R[100]mm/sec CNT100;
   1:  PR[91,1] = PR[90,1] + -88.011;
   1:  PR[91,2] = PR[90,2] + -17.471;
   1:L PR[91] R[100]mm/sec CNT100;
   1:  PR[91,1] = PR[90,1] + -87.398;
   1:  PR[91,2] = PR[90,2] + -17.693;
   1:L PR[91] R[100]mm/sec CNT100;
   1:  PR[91,1] = PR[90,1] + -87.093;
   1:  PR[91,2] = PR[90,2] + -18.319;
   1:L PR[91] R[100]mm/sec CNT100;
   1:  PR[91,1] = PR[90,1] + -87.081;
   1:  PR[91,2] = PR[90,2] + -18.337;
   1:L PR[91] R[100]mm/sec CNT100;
   1:  PR[91,1] = PR[90,1] + -87.055;
   1:  PR[91,2] = PR[90,2] + -18.350;
   1:L PR[91] R[100]mm/sec CNT100;
   1:  PR[91,1] = PR[90,1] + -86.409;
   1:  PR[91,2] = PR[90,2] + -18.602;
   1:L PR[91] R[100]mm/sec CNT100;
   1:  PR[91,1] = PR[90,1] + -86.014;
   1:  PR[91,2] = PR[90,2] + -19.193;
   1:L PR[91] R[100]mm/sec CNT100;
   1:  PR[91,1] = PR[90,1] + -85.450;
   1:  PR[91,2] = PR[90,2] + -19.480;
   1:L PR[91] R[100]mm/sec CNT100;
   1:  PR[91,1] = PR[90,1] + -84.837;
   1:  PR[91,2] = PR[90,2] + -20.003;
   1:L PR[91] R[100]mm/sec CNT100;
   1:  PR[91,1] = PR[90,1] + -84.396;
   1:  PR[91,2] = PR[90,2] + -20.342;
   1:L PR[91] R[100]mm/sec CNT100;
   1:  PR[91,1] = PR[90,1] + -84.153;
   1:  PR[91,2] = PR[90,2] + -20.452;
   1:L PR[91] R[100]mm/sec CNT100;
   1:  PR[91,1] = PR[90,1] + -83.642;
   1:  PR[91,2] = PR[90,2] + -20.574;
   1:L PR[91] R[100]mm/sec CNT100;
   1:  PR[91,1] = PR[90,1] + -83.155;
   1:  PR[91,2] = PR[90,2] + -21.125;
   1:L PR[91] R[100]mm/sec CNT100;
   1:  PR[91,1] = PR[90,1] + -83.138;
   1:  PR[91,2] = PR[90,2] + -21.130;
   1:L PR[91] R[100]mm/sec CNT100;
   1:  PR[91,1] = PR[90,1] + -82.605;
   1:  PR[91,2] = PR[90,2] + -21.364;
   1:L PR[91] R[100]mm/sec CNT100;
   1:  PR[91,1] = PR[90,1] + -82.161;
   1:  PR[91,2] = PR[90,2] + -21.582;
   1:L PR[91] R[100]mm/sec CNT100;
   1:  PR[91,1] = PR[90,1] + -81.793;
   1:  PR[91,2] = PR[90,2] + -21.646;
   1:L PR[91] R[100]mm/sec CNT100;
   1:  PR[91,1] = PR[90,1] + -81.428;
   1:  PR[91,2] = PR[90,2] + -22.033;
   1:L PR[91] R[100]mm/sec CNT100;
   1:  PR[91,1] = PR[90,1] + -81.318;
   1:  PR[91,2] = PR[90,2] + -22.127;
   1:L PR[91] R[100]mm/sec CNT100;
   1:  PR[91,1] = PR[90,1] + -81.199;
   1:  PR[91,2] = PR[90,2] + -22.154;
   1:L PR[91] R[100]mm/sec CNT100;
   1:  PR[91,1] = PR[90,1] + -80.249;
   1:  PR[91,2] = PR[90,2] + -22.502;
   1:L PR[91] R[100]mm/sec CNT100;
   1:  PR[91,1] = PR[90,1] + -79.878;
   1:  PR[91,2] = PR[90,2] + -22.556;
   1:L PR[91] R[100]mm/sec CNT100;
   1:  PR[91,1] = PR[90,1] + -79.285;
   1:  PR[91,2] = PR[90,2] + -22.997;
   1:L PR[91] R[100]mm/sec CNT100;
   1:  PR[91,1] = PR[90,1] + -79.195;
   1:  PR[91,2] = PR[90,2] + -23.012;
   1:L PR[91] R[100]mm/sec CNT100;
   1:  PR[91,1] = PR[90,1] + -78.708;
   1:  PR[91,2] = PR[90,2] + -23.215;
   1:L PR[91] R[100]mm/sec CNT100;
   1:  PR[91,1] = PR[90,1] + -77.908;
   1:  PR[91,2] = PR[90,2] + -23.358;
   1:L PR[91] R[100]mm/sec CNT100;
   1:  PR[91,1] = PR[90,1] + -77.290;
   1:  PR[91,2] = PR[90,2] + -23.564;
   1:L PR[91] R[100]mm/sec CNT100;
   1:  PR[91,1] = PR[90,1] + -77.091;
   1:  PR[91,2] = PR[90,2] + -23.584;
   1:L PR[91] R[100]mm/sec CNT100;
   1:  PR[91,1] = PR[90,1] + -76.396;
   1:  PR[91,2] = PR[90,2] + -23.923;
   1:L PR[91] R[100]mm/sec CNT100;
   1:  PR[91,1] = PR[90,1] + -76.273;
   1:  PR[91,2] = PR[90,2] + -23.939;
   1:L PR[91] R[100]mm/sec CNT100;
   1:  PR[91,1] = PR[90,1] + -75.729;
   1:  PR[91,2] = PR[90,2] + -24.114;
   1:L PR[91] R[100]mm/sec CNT100;
   1:  PR[91,1] = PR[90,1] + -75.372;
   1:  PR[91,2] = PR[90,2] + -24.149;
   1:L PR[91] R[100]mm/sec CNT100;
   1:  PR[91,1] = PR[90,1] + -74.941;
   1:  PR[91,2] = PR[90,2] + -24.237;
   1:L PR[91] R[100]mm/sec CNT100;
   1:  PR[91,1] = PR[90,1] + -74.066;
   1:  PR[91,2] = PR[90,2] + -24.318;
   1:L PR[91] R[100]mm/sec CNT100;
   1:  PR[91,1] = PR[90,1] + -73.449;
   1:  PR[91,2] = PR[90,2] + -24.405;
   1:L PR[91] R[100]mm/sec CNT100;
   1:  PR[91,1] = PR[90,1] + -73.200;
   1:  PR[91,2] = PR[90,2] + -24.415;
   1:L PR[91] R[100]mm/sec CNT100;
   1:  PR[91,1] = PR[90,1] + -72.397;
   1:  PR[91,2] = PR[90,2] + -24.531;
   1:L PR[91] R[100]mm/sec CNT100;
   1:  PR[91,1] = PR[90,1] + -71.443;
   1:  PR[91,2] = PR[90,2] + -24.627;
   1:L PR[91] R[100]mm/sec CNT100;
   1:  PR[91,1] = PR[90,1] + -70.534;
   1:  PR[91,2] = PR[90,2] + -24.695;
   1:L PR[91] R[100]mm/sec CNT100;
   1:  PR[91,1] = PR[90,1] + -69.591;
   1:  PR[91,2] = PR[90,2] + -24.713;
   1:L PR[91] R[100]mm/sec CNT100;
   1:  PR[91,1] = PR[90,1] + -68.668;
   1:  PR[91,2] = PR[90,2] + -24.663;
   1:L PR[91] R[100]mm/sec CNT100;
   1:  PR[91,1] = PR[90,1] + -67.623;
   1:  PR[91,2] = PR[90,2] + -24.569;
   1:L PR[91] R[100]mm/sec CNT100;
   1:  PR[91,1] = PR[90,1] + -66.710;
   1:  PR[91,2] = PR[90,2] + -24.447;
   1:L PR[91] R[100]mm/sec CNT100;
   1:  PR[91,1] = PR[90,1] + -66.476;
   1:  PR[91,2] = PR[90,2] + -24.427;
   1:L PR[91] R[100]mm/sec CNT100;
   1:  PR[91,1] = PR[90,1] + -65.793;
   1:  PR[91,2] = PR[90,2] + -24.331;
   1:L PR[91] R[100]mm/sec CNT100;
   1:  PR[91,1] = PR[90,1] + -65.345;
   1:  PR[91,2] = PR[90,2] + -24.244;
   1:L PR[91] R[100]mm/sec CNT100;
   1:  PR[91,1] = PR[90,1] + -64.841;
   1:  PR[91,2] = PR[90,2] + -24.185;
   1:L PR[91] R[100]mm/sec CNT100;
   1:  PR[91,1] = PR[90,1] + -64.148;
   1:  PR[91,2] = PR[90,2] + -23.980;
   1:L PR[91] R[100]mm/sec CNT100;
   1:  PR[91,1] = PR[90,1] + -63.922;
   1:  PR[91,2] = PR[90,2] + -23.951;
   1:L PR[91] R[100]mm/sec CNT100;
   1:  PR[91,1] = PR[90,1] + -63.424;
   1:  PR[91,2] = PR[90,2] + -23.747;
   1:L PR[91] R[100]mm/sec CNT100;
   1:  PR[91,1] = PR[90,1] + -62.983;
   1:  PR[91,2] = PR[90,2] + -23.589;
   1:L PR[91] R[100]mm/sec CNT100;
   1:  PR[91,1] = PR[90,1] + -62.012;
   1:  PR[91,2] = PR[90,2] + -23.319;
   1:L PR[91] R[100]mm/sec CNT100;
   1:  PR[91,1] = PR[90,1] + -61.299;
   1:  PR[91,2] = PR[90,2] + -23.026;
   1:L PR[91] R[100]mm/sec CNT100;
   1:  PR[91,1] = PR[90,1] + -61.067;
   1:  PR[91,2] = PR[90,2] + -22.972;
   1:L PR[91] R[100]mm/sec CNT100;
   1:  PR[91,1] = PR[90,1] + -60.751;
   1:  PR[91,2] = PR[90,2] + -22.795;
   1:L PR[91] R[100]mm/sec CNT100;
   1:  PR[91,1] = PR[90,1] + -60.123;
   1:  PR[91,2] = PR[90,2] + -22.513;
   1:L PR[91] R[100]mm/sec CNT100;
   1:  PR[91,1] = PR[90,1] + -59.618;
   1:  PR[91,2] = PR[90,2] + -22.292;
   1:L PR[91] R[100]mm/sec CNT100;
   1:  PR[91,1] = PR[90,1] + -59.159;
   1:  PR[91,2] = PR[90,2] + -22.132;
   1:L PR[91] R[100]mm/sec CNT100;
   1:  PR[91,1] = PR[90,1] + -58.675;
   1:  PR[91,2] = PR[90,2] + -21.831;
   1:L PR[91] R[100]mm/sec CNT100;
   1:  PR[91,1] = PR[90,1] + -58.220;
   1:  PR[91,2] = PR[90,2] + -21.578;
   1:L PR[91] R[100]mm/sec CNT100;
   1:  PR[91,1] = PR[90,1] + -57.677;
   1:  PR[91,2] = PR[90,2] + -21.290;
   1:L PR[91] R[100]mm/sec CNT100;
   1:  PR[91,1] = PR[90,1] + -57.242;
   1:  PR[91,2] = PR[90,2] + -21.100;
   1:L PR[91] R[100]mm/sec CNT100;
   1:  PR[91,1] = PR[90,1] + -56.902;
   1:  PR[91,2] = PR[90,2] + -20.858;
   1:L PR[91] R[100]mm/sec CNT100;
   1:  PR[91,1] = PR[90,1] + -56.302;
   1:  PR[91,2] = PR[90,2] + -20.496;
   1:L PR[91] R[100]mm/sec CNT100;
   1:  PR[91,1] = PR[90,1] + -55.310;
   1:  PR[91,2] = PR[90,2] + -19.827;
   1:L PR[91] R[100]mm/sec CNT100;
   1:  PR[91,1] = PR[90,1] + -54.369;
   1:  PR[91,2] = PR[90,2] + -19.230;
   1:L PR[91] R[100]mm/sec CNT100;
   1:  PR[91,1] = PR[90,1] + -53.992;
   1:  PR[91,2] = PR[90,2] + -18.917;
   1:L PR[91] R[100]mm/sec CNT100;
   1:  PR[91,1] = PR[90,1] + -53.427;
   1:  PR[91,2] = PR[90,2] + -18.484;
   1:L PR[91] R[100]mm/sec CNT100;
   1:  PR[91,1] = PR[90,1] + -52.471;
   1:  PR[91,2] = PR[90,2] + -17.658;
   1:L PR[91] R[100]mm/sec CNT100;
   1:  PR[91,1] = PR[90,1] + -51.500;
   1:  PR[91,2] = PR[90,2] + -16.770;
   1:L PR[91] R[100]mm/sec CNT100;
   1:  PR[91,1] = PR[90,1] + -50.532;
   1:  PR[91,2] = PR[90,2] + -15.822;
   1:L PR[91] R[100]mm/sec CNT100;
   1:  PR[91,1] = PR[90,1] + -49.773;
   1:  PR[91,2] = PR[90,2] + -15.025;
   1:L PR[91] R[100]mm/sec CNT100;
   1:  PR[91,1] = PR[90,1] + -48.585;
   1:  PR[91,2] = PR[90,2] + -13.697;
   1:L PR[91] R[100]mm/sec CNT100;
   1:  PR[91,1] = PR[90,1] + -48.049;
   1:  PR[91,2] = PR[90,2] + -13.066;
   1:L PR[91] R[100]mm/sec CNT100;
   1:  PR[91,1] = PR[90,1] + -47.291;
   1:  PR[91,2] = PR[90,2] + -12.118;
   1:L PR[91] R[100]mm/sec CNT100;
   1:  PR[91,1] = PR[90,1] + -46.651;
   1:  PR[91,2] = PR[90,2] + -11.172;
   1:L PR[91] R[100]mm/sec CNT100;
   1:  PR[91,1] = PR[90,1] + -45.999;
   1:  PR[91,2] = PR[90,2] + -10.151;
   1:L PR[91] R[100]mm/sec CNT100;
   1:  PR[92] = PR[91];
   1:  PR[92,3] = PR[92,3] + R[101];
   1:J PR[92] R[102]% CNT100;
   1:  PR[91,1] = PR[90,1] + -55.042;
   1:  PR[91,2] = PR[90,2] + -5.607;
   1:  PR[92] = PR[91];
   1:  PR[92,3] = PR[92,3] + R[101];
   1:J PR[92] R[102]% CNT100;
   1:L PR[91] 100mm/sec CNT100 RampTo R[100];
   1:  PR[91,1] = PR[90,1] + -56.292;
   1:  PR[91,2] = PR[90,2] + -7.524;
   1:L PR[91] R[100]mm/sec CNT100;
   1:  PR[91,1] = PR[90,1] + -56.575;
   1:  PR[91,2] = PR[90,2] + -7.869;
   1:L PR[91] R[100]mm/sec CNT100;
   1:  PR[91,1] = PR[90,1] + -57.376;
   1:  PR[91,2] = PR[90,2] + -8.918;
   1:L PR[91] R[100]mm/sec CNT100;
   1:  PR[91,1] = PR[90,1] + -58.537;
   1:  PR[91,2] = PR[90,2] + -10.087;
   1:L PR[91] R[100]mm/sec CNT100;
   1:  PR[91,1] = PR[90,1] + -59.574;
   1:  PR[91,2] = PR[90,2] + -10.892;
   1:L PR[91] R[100]mm/sec CNT100;
   1:  PR[91,1] = PR[90,1] + -59.905;
   1:  PR[91,2] = PR[90,2] + -11.173;
   1:L PR[91] R[100]mm/sec CNT100;
   1:  PR[91,1] = PR[90,1] + -61.821;
   1:  PR[91,2] = PR[90,2] + -12.448;
   1:L PR[91] R[100]mm/sec CNT100;
   1:  PR[91,1] = PR[90,1] + -62.925;
   1:  PR[91,2] = PR[90,2] + -12.903;
   1:L PR[91] R[100]mm/sec CNT100;
   1:  PR[91,1] = PR[90,1] + -63.979;
   1:  PR[91,2] = PR[90,2] + -13.405;
   1:L PR[91] R[100]mm/sec CNT100;
   1:  PR[91,1] = PR[90,1] + -65.168;
   1:  PR[91,2] = PR[90,2] + -13.799;
   1:L PR[91] R[100]mm/sec CNT100;
   1:  PR[91,1] = PR[90,1] + -67.011;
   1:  PR[91,2] = PR[90,2] + -14.145;
   1:L PR[91] R[100]mm/sec CNT100;
   1:  PR[91,1] = PR[90,1] + -67.386;
   1:  PR[91,2] = PR[90,2] + -14.172;
   1:L PR[91] R[100]mm/sec CNT100;
   1:  PR[91,1] = PR[90,1] + -68.205;
   1:  PR[91,2] = PR[90,2] + -14.298;
   1:L PR[91] R[100]mm/sec CNT100;
   1:  PR[91,1] = PR[90,1] + -69.547;
   1:  PR[91,2] = PR[90,2] + -14.366;
   1:L PR[91] R[100]mm/sec CNT100;
   1:  PR[91,1] = PR[90,1] + -70.692;
   1:  PR[91,2] = PR[90,2] + -14.335;
   1:L PR[91] R[100]mm/sec CNT100;
   1:  PR[91,1] = PR[90,1] + -71.434;
   1:  PR[91,2] = PR[90,2] + -14.234;
   1:L PR[91] R[100]mm/sec CNT100;
   1:  PR[91,1] = PR[90,1] + -71.766;
   1:  PR[91,2] = PR[90,2] + -14.222;
   1:L PR[91] R[100]mm/sec CNT100;
   1:  PR[91,1] = PR[90,1] + -72.377;
   1:  PR[91,2] = PR[90,2] + -14.085;
   1:L PR[91] R[100]mm/sec CNT100;
   1:  PR[91,1] = PR[90,1] + -72.808;
   1:  PR[91,2] = PR[90,2] + -14.060;
   1:L PR[91] R[100]mm/sec CNT100;
   1:  PR[91,1] = PR[90,1] + -73.296;
   1:  PR[91,2] = PR[90,2] + -13.937;
   1:L PR[91] R[100]mm/sec CNT100;
   1:  PR[91,1] = PR[90,1] + -73.790;
   1:  PR[91,2] = PR[90,2] + -13.888;
   1:L PR[91] R[100]mm/sec CNT100;
   1:  PR[91,1] = PR[90,1] + -74.271;
   1:  PR[91,2] = PR[90,2] + -13.803;
   1:L PR[91] R[100]mm/sec CNT100;
   1:  PR[91,1] = PR[90,1] + -74.922;
   1:  PR[91,2] = PR[90,2] + -13.610;
   1:L PR[91] R[100]mm/sec CNT100;
   1:  PR[91,1] = PR[90,1] + -75.243;
   1:  PR[91,2] = PR[90,2] + -13.559;
   1:L PR[91] R[100]mm/sec CNT100;
   1:  PR[91,1] = PR[90,1] + -75.790;
   1:  PR[91,2] = PR[90,2] + -13.227;
   1:L PR[91] R[100]mm/sec CNT100;
   1:  PR[91,1] = PR[90,1] + -75.922;
   1:  PR[91,2] = PR[90,2] + -13.120;
   1:L PR[91] R[100]mm/sec CNT100;
   1:  PR[91,1] = PR[90,1] + -76.065;
   1:  PR[91,2] = PR[90,2] + -13.099;
   1:L PR[91] R[100]mm/sec CNT100;
   1:  PR[91,1] = PR[90,1] + -76.583;
   1:  PR[91,2] = PR[90,2] + -12.829;
   1:L PR[91] R[100]mm/sec CNT100;
   1:  PR[91,1] = PR[90,1] + -77.531;
   1:  PR[91,2] = PR[90,2] + -12.569;
   1:L PR[91] R[100]mm/sec CNT100;
   1:  PR[91,1] = PR[90,1] + -78.174;
   1:  PR[91,2] = PR[90,2] + -12.035;
   1:L PR[91] R[100]mm/sec CNT100;
   1:  PR[91,1] = PR[90,1] + -78.181;
   1:  PR[91,2] = PR[90,2] + -12.034;
   1:L PR[91] R[100]mm/sec CNT100;
   1:  PR[91,1] = PR[90,1] + -78.753;
   1:  PR[91,2] = PR[90,2] + -11.666;
   1:L PR[91] R[100]mm/sec CNT100;
   1:  PR[91,1] = PR[90,1] + -79.650;
   1:  PR[91,2] = PR[90,2] + -11.196;
   1:L PR[91] R[100]mm/sec CNT100;
   1:  PR[91,1] = PR[90,1] + -80.053;
   1:  PR[91,2] = PR[90,2] + -10.666;
   1:L PR[91] R[100]mm/sec CNT100;
   1:  PR[91,1] = PR[90,1] + -80.836;
   1:  PR[91,2] = PR[90,2] + -10.322;
   1:L PR[91] R[100]mm/sec CNT100;
   1:  PR[91,1] = PR[90,1] + -81.216;
   1:  PR[91,2] = PR[90,2] + -9.686;
   1:L PR[91] R[100]mm/sec CNT100;
   1:  PR[91,1] = PR[90,1] + -81.250;
   1:  PR[91,2] = PR[90,2] + -9.619;
   1:L PR[91] R[100]mm/sec CNT100;
   1:  PR[91,1] = PR[90,1] + -81.320;
   1:  PR[91,2] = PR[90,2] + -9.586;
   1:L PR[91] R[100]mm/sec CNT100;
   1:  PR[91,1] = PR[90,1] + -81.994;
   1:  PR[91,2] = PR[90,2] + -9.192;
   1:L PR[91] R[100]mm/sec CNT100;
   1:  PR[91,1] = PR[90,1] + -82.315;
   1:  PR[91,2] = PR[90,2] + -8.453;
   1:L PR[91] R[100]mm/sec CNT100;
   1:  PR[91,1] = PR[90,1] + -82.995;
   1:  PR[91,2] = PR[90,2] + -8.011;
   1:L PR[91] R[100]mm/sec CNT100;
   1:  PR[91,1] = PR[90,1] + -83.164;
   1:  PR[91,2] = PR[90,2] + -7.486;
   1:L PR[91] R[100]mm/sec CNT100;
   1:  PR[91,1] = PR[90,1] + -83.321;
   1:  PR[91,2] = PR[90,2] + -7.148;
   1:L PR[91] R[100]mm/sec CNT100;
   1:  PR[91,1] = PR[90,1] + -83.654;
   1:  PR[91,2] = PR[90,2] + -6.742;
   1:L PR[91] R[100]mm/sec CNT100;
   1:  PR[91,1] = PR[90,1] + -83.664;
   1:  PR[91,2] = PR[90,2] + -6.736;
   1:L PR[91] R[100]mm/sec CNT100;
   1:  PR[91,1] = PR[90,1] + -83.698;
   1:  PR[91,2] = PR[90,2] + -6.688;
   1:L PR[91] R[100]mm/sec CNT100;
   1:  PR[91,1] = PR[90,1] + -83.776;
   1:  PR[91,2] = PR[90,2] + -6.592;
   1:L PR[91] R[100]mm/sec CNT100;
   1:  PR[91,1] = PR[90,1] + -83.781;
   1:  PR[91,2] = PR[90,2] + -6.572;
   1:L PR[91] R[100]mm/sec CNT100;
   1:  PR[91,1] = PR[90,1] + -84.269;
   1:  PR[91,2] = PR[90,2] + -5.887;
   1:L PR[91] R[100]mm/sec CNT100;
   1:  PR[91,1] = PR[90,1] + -84.460;
   1:  PR[91,2] = PR[90,2] + -5.306;
   1:L PR[91] R[100]mm/sec CNT100;
   1:  PR[91,1] = PR[90,1] + -84.520;
   1:  PR[91,2] = PR[90,2] + -5.026;
   1:L PR[91] R[100]mm/sec CNT100;
   1:  PR[91,1] = PR[90,1] + -84.849;
   1:  PR[91,2] = PR[90,2] + -4.580;
   1:L PR[91] R[100]mm/sec CNT100;
   1:  PR[91,1] = PR[90,1] + -84.912;
   1:  PR[91,2] = PR[90,2] + -4.496;
   1:L PR[91] R[100]mm/sec CNT100;
   1:  PR[91,1] = PR[90,1] + -84.920;
   1:  PR[91,2] = PR[90,2] + -4.438;
   1:L PR[91] R[100]mm/sec CNT100;
   1:  PR[91,1] = PR[90,1] + -85.324;
   1:  PR[91,2] = PR[90,2] + -3.629;
   1:L PR[91] R[100]mm/sec CNT100;
   1:  PR[91,1] = PR[90,1] + -85.507;
   1:  PR[91,2] = PR[90,2] + -2.653;
   1:L PR[91] R[100]mm/sec CNT100;
   1:  PR[91,1] = PR[90,1] + -85.656;
   1:  PR[91,2] = PR[90,2] + -2.163;
   1:L PR[91] R[100]mm/sec CNT100;
   1:  PR[91,1] = PR[90,1] + -85.688;
   1:  PR[91,2] = PR[90,2] + -1.776;
   1:L PR[91] R[100]mm/sec CNT100;
   1:  PR[91,1] = PR[90,1] + -85.908;
   1:  PR[91,2] = PR[90,2] + -1.184;
   1:L PR[91] R[100]mm/sec CNT100;
   1:  PR[91,1] = PR[90,1] + -85.924;
   1:  PR[91,2] = PR[90,2] + -0.944;
   1:L PR[91] R[100]mm/sec CNT100;
   1:  PR[91,1] = PR[90,1] + -86.151;
   1:  PR[91,2] = PR[90,2] + -0.221;
   1:L PR[91] R[100]mm/sec CNT100;
   1:  PR[91,1] = PR[90,1] + -86.293;
   1:  PR[91,2] = PR[90,2] + 0.867;
   1:L PR[91] R[100]mm/sec CNT100;
   1:  PR[91,1] = PR[90,1] + -86.350;
   1:  PR[91,2] = PR[90,2] + 2.157;
   1:L PR[91] R[100]mm/sec CNT100;
   1:  PR[91,1] = PR[90,1] + -86.316;
   1:  PR[91,2] = PR[90,2] + 3.283;
   1:L PR[91] R[100]mm/sec CNT100;
   1:  PR[91,1] = PR[90,1] + -86.189;
   1:  PR[91,2] = PR[90,2] + 4.448;
   1:L PR[91] R[100]mm/sec CNT100;
   1:  PR[91,1] = PR[90,1] + -85.950;
   1:  PR[91,2] = PR[90,2] + 5.446;
   1:L PR[91] R[100]mm/sec CNT100;
   1:  PR[91,1] = PR[90,1] + -85.930;
   1:  PR[91,2] = PR[90,2] + 5.665;
   1:L PR[91] R[100]mm/sec CNT100;
   1:  PR[91,1] = PR[90,1] + -85.683;
   1:  PR[91,2] = PR[90,2] + 6.556;
   1:L PR[91] R[100]mm/sec CNT100;
   1:  PR[91,1] = PR[90,1] + -85.586;
   1:  PR[91,2] = PR[90,2] + 7.064;
   1:L PR[91] R[100]mm/sec CNT100;
   1:  PR[91,1] = PR[90,1] + -85.423;
   1:  PR[91,2] = PR[90,2] + 7.698;
   1:L PR[91] R[100]mm/sec CNT100;
   1:  PR[91,1] = PR[90,1] + -84.918;
   1:  PR[91,2] = PR[90,2] + 8.938;
   1:L PR[91] R[100]mm/sec CNT100;
   1:  PR[91,1] = PR[90,1] + -84.429;
   1:  PR[91,2] = PR[90,2] + 9.934;
   1:L PR[91] R[100]mm/sec CNT100;
   1:  PR[91,1] = PR[90,1] + -83.900;
   1:  PR[91,2] = PR[90,2] + 10.924;
   1:L PR[91] R[100]mm/sec CNT100;
   1:  PR[91,1] = PR[90,1] + -83.787;
   1:  PR[91,2] = PR[90,2] + 11.076;
   1:L PR[91] R[100]mm/sec CNT100;
   1:  PR[91,1] = PR[90,1] + -83.675;
   1:  PR[91,2] = PR[90,2] + 11.277;
   1:L PR[91] R[100]mm/sec CNT100;
   1:  PR[91,1] = PR[90,1] + -83.106;
   1:  PR[91,2] = PR[90,2] + 12.151;
   1:L PR[91] R[100]mm/sec CNT100;
   1:  PR[91,1] = PR[90,1] + -82.782;
   1:  PR[91,2] = PR[90,2] + 12.557;
   1:L PR[91] R[100]mm/sec CNT100;
   1:  PR[91,1] = PR[90,1] + -82.168;
   1:  PR[91,2] = PR[90,2] + 13.277;
   1:L PR[91] R[100]mm/sec CNT100;
   1:  PR[91,1] = PR[90,1] + -81.705;
   1:  PR[91,2] = PR[90,2] + 13.784;
   1:L PR[91] R[100]mm/sec CNT100;
   1:  PR[91,1] = PR[90,1] + -81.114;
   1:  PR[91,2] = PR[90,2] + 14.376;
   1:L PR[91] R[100]mm/sec CNT100;
   1:  PR[91,1] = PR[90,1] + -80.614;
   1:  PR[91,2] = PR[90,2] + 14.839;
   1:L PR[91] R[100]mm/sec CNT100;
   1:  PR[91,1] = PR[90,1] + -79.889;
   1:  PR[91,2] = PR[90,2] + 15.463;
   1:L PR[91] R[100]mm/sec CNT100;
   1:  PR[91,1] = PR[90,1] + -79.501;
   1:  PR[91,2] = PR[90,2] + 15.772;
   1:L PR[91] R[100]mm/sec CNT100;
   1:  PR[91,1] = PR[90,1] + -78.614;
   1:  PR[91,2] = PR[90,2] + 16.378;
   1:L PR[91] R[100]mm/sec CNT100;
   1:  PR[91,1] = PR[90,1] + -78.419;
   1:  PR[91,2] = PR[90,2] + 16.489;
   1:L PR[91] R[100]mm/sec CNT100;
   1:  PR[91,1] = PR[90,1] + -78.267;
   1:  PR[91,2] = PR[90,2] + 16.599;
   1:L PR[91] R[100]mm/sec CNT100;
   1:  PR[91,1] = PR[90,1] + -76.317;
   1:  PR[91,2] = PR[90,2] + 17.615;
   1:L PR[91] R[100]mm/sec CNT100;
   1:  PR[91,1] = PR[90,1] + -76.088;
   1:  PR[91,2] = PR[90,2] + 17.721;
   1:L PR[91] R[100]mm/sec CNT100;
   1:  PR[91,1] = PR[90,1] + -75.054;
   1:  PR[91,2] = PR[90,2] + 18.093;
   1:L PR[91] R[100]mm/sec CNT100;
   1:  PR[91,1] = PR[90,1] + -74.475;
   1:  PR[91,2] = PR[90,2] + 18.261;
   1:L PR[91] R[100]mm/sec CNT100;
   1:  PR[91,1] = PR[90,1] + -73.935;
   1:  PR[91,2] = PR[90,2] + 18.367;
   1:L PR[91] R[100]mm/sec CNT100;
   1:  PR[91,1] = PR[90,1] + -73.095;
   1:  PR[91,2] = PR[90,2] + 18.607;
   1:L PR[91] R[100]mm/sec CNT100;
   1:  PR[91,1] = PR[90,1] + -72.860;
   1:  PR[91,2] = PR[90,2] + 18.639;
   1:L PR[91] R[100]mm/sec CNT100;
   1:  PR[91,1] = PR[90,1] + -72.177;
   1:  PR[91,2] = PR[90,2] + 18.806;
   1:L PR[91] R[100]mm/sec CNT100;
   1:  PR[91,1] = PR[90,1] + -71.804;
   1:  PR[91,2] = PR[90,2] + 18.883;
   1:L PR[91] R[100]mm/sec CNT100;
   1:  PR[91,1] = PR[90,1] + -70.662;
   1:  PR[91,2] = PR[90,2] + 19.002;
   1:L PR[91] R[100]mm/sec CNT100;
   1:  PR[91,1] = PR[90,1] + -69.357;
   1:  PR[91,2] = PR[90,2] + 19.027;
   1:L PR[91] R[100]mm/sec CNT100;
   1:  PR[91,1] = PR[90,1] + -68.274;
   1:  PR[91,2] = PR[90,2] + 18.970;
   1:L PR[91] R[100]mm/sec CNT100;
   1:  PR[91,1] = PR[90,1] + -67.212;
   1:  PR[91,2] = PR[90,2] + 18.809;
   1:L PR[91] R[100]mm/sec CNT100;
   1:  PR[91,1] = PR[90,1] + -66.496;
   1:  PR[91,2] = PR[90,2] + 18.587;
   1:L PR[91] R[100]mm/sec CNT100;
   1:  PR[91,1] = PR[90,1] + -66.239;
   1:  PR[91,2] = PR[90,2] + 18.565;
   1:L PR[91] R[100]mm/sec CNT100;
   1:  PR[91,1] = PR[90,1] + -65.656;
   1:  PR[91,2] = PR[90,2] + 18.366;
   1:L PR[91] R[100]mm/sec CNT100;
   1:  PR[91,1] = PR[90,1] + -65.273;
   1:  PR[91,2] = PR[90,2] + 18.321;
   1:L PR[91] R[100]mm/sec CNT100;
   1:  PR[91,1] = PR[90,1] + -64.251;
   1:  PR[91,2] = PR[90,2] + 18.063;
   1:L PR[91] R[100]mm/sec CNT100;
   1:  PR[91,1] = PR[90,1] + -63.789;
   1:  PR[91,2] = PR[90,2] + 17.999;
   1:L PR[91] R[100]mm/sec CNT100;
   1:  PR[91,1] = PR[90,1] + -63.059;
   1:  PR[91,2] = PR[90,2] + 17.541;
   1:L PR[91] R[100]mm/sec CNT100;
   1:  PR[91,1] = PR[90,1] + -63.053;
   1:  PR[91,2] = PR[90,2] + 17.536;
   1:L PR[91] R[100]mm/sec CNT100;
   1:  PR[91,1] = PR[90,1] + -62.999;
   1:  PR[91,2] = PR[90,2] + 17.526;
   1:L PR[91] R[100]mm/sec CNT100;
   1:  PR[91,1] = PR[90,1] + -62.431;
   1:  PR[91,2] = PR[90,2] + 17.192;
   1:L PR[91] R[100]mm/sec CNT100;
   1:  PR[91,1] = PR[90,1] + -62.124;
   1:  PR[91,2] = PR[90,2] + 17.095;
   1:L PR[91] R[100]mm/sec CNT100;
   1:  PR[91,1] = PR[90,1] + -61.529;
   1:  PR[91,2] = PR[90,2] + 16.948;
   1:L PR[91] R[100]mm/sec CNT100;
   1:  PR[91,1] = PR[90,1] + -60.920;
   1:  PR[91,2] = PR[90,2] + 16.383;
   1:L PR[91] R[100]mm/sec CNT100;
   1:  PR[91,1] = PR[90,1] + -60.903;
   1:  PR[91,2] = PR[90,2] + 16.378;
   1:L PR[91] R[100]mm/sec CNT100;
   1:  PR[91,1] = PR[90,1] + -59.927;
   1:  PR[91,2] = PR[90,2] + 15.753;
   1:L PR[91] R[100]mm/sec CNT100;
   1:  PR[91,1] = PR[90,1] + -59.404;
   1:  PR[91,2] = PR[90,2] + 15.630;
   1:L PR[91] R[100]mm/sec CNT100;
   1:  PR[91,1] = PR[90,1] + -59.188;
   1:  PR[91,2] = PR[90,2] + 15.126;
   1:L PR[91] R[100]mm/sec CNT100;
   1:  PR[91,1] = PR[90,1] + -59.045;
   1:  PR[91,2] = PR[90,2] + 14.966;
   1:L PR[91] R[100]mm/sec CNT100;
   1:  PR[91,1] = PR[90,1] + -58.874;
   1:  PR[91,2] = PR[90,2] + 14.861;
   1:L PR[91] R[100]mm/sec CNT100;
   1:  PR[91,1] = PR[90,1] + -58.227;
   1:  PR[91,2] = PR[90,2] + 14.643;
   1:L PR[91] R[100]mm/sec CNT100;
   1:  PR[91,1] = PR[90,1] + -57.972;
   1:  PR[91,2] = PR[90,2] + 13.997;
   1:L PR[91] R[100]mm/sec CNT100;
   1:  PR[91,1] = PR[90,1] + -57.888;
   1:  PR[91,2] = PR[90,2] + 13.870;
   1:L PR[91] R[100]mm/sec CNT100;
   1:  PR[91,1] = PR[90,1] + -57.768;
   1:  PR[91,2] = PR[90,2] + 13.783;
   1:L PR[91] R[100]mm/sec CNT100;
   1:  PR[91,1] = PR[90,1] + -57.147;
   1:  PR[91,2] = PR[90,2] + 13.524;
   1:L PR[91] R[100]mm/sec CNT100;
   1:  PR[91,1] = PR[90,1] + -56.961;
   1:  PR[91,2] = PR[90,2] + 12.901;
   1:L PR[91] R[100]mm/sec CNT100;
   1:  PR[91,1] = PR[90,1] + -56.822;
   1:  PR[91,2] = PR[90,2] + 12.675;
   1:L PR[91] R[100]mm/sec CNT100;
   1:  PR[91,1] = PR[90,1] + -56.549;
   1:  PR[91,2] = PR[90,2] + 12.381;
   1:L PR[91] R[100]mm/sec CNT100;
   1:  PR[91,1] = PR[90,1] + -56.485;
   1:  PR[91,2] = PR[90,2] + 12.346;
   1:L PR[91] R[100]mm/sec CNT100;
   1:  PR[91,1] = PR[90,1] + -56.378;
   1:  PR[91,2] = PR[90,2] + 12.198;
   1:L PR[91] R[100]mm/sec CNT100;
   1:  PR[91,1] = PR[90,1] + -56.199;
   1:  PR[91,2] = PR[90,2] + 12.005;
   1:L PR[91] R[100]mm/sec CNT100;
   1:  PR[91,1] = PR[90,1] + -56.179;
